	UF : 0, UT : 6,		CONFIG : 'N U T, 0, 0, 0',
	X =  493.676  mm,	Y =   -406.000  mm,	Z =   -242.674  mm,
	W =  90.000 deg,	P =   0.000 deg,	R =   90.000 deg
};
P[579]{
   GP1:
	UF : 0, UT : 6,		CONFIG : 'N U T, 0, 0, 0',
	X =  491.508  mm,	Y =   -402.493  mm,	Z =   -243.023  mm,
	W =  90.000 deg,	P =   0.000 deg,	R =   90.000 deg
};
P[580]{
   GP1:
	UF : 0, UT : 6,		CONFIG : 'N U T, 0, 0, 0',
	X =  491.035  mm,	Y =   -401.706  mm,	Z =   -243.069  mm,
	W =  90.000 deg,	P =   0.000 deg,	R =   90.000 deg
};
P[581]{
   GP1:
	UF : 0, UT : 6,		CONFIG : 'N U T, 0, 0, 0',
	X =  488.683  mm,	Y =   -397.423  mm,	Z =   -242.773  mm,
	W =  90.000 deg,	P =   0.000 deg,	R =   90.000 deg
};
P[582]{
   GP1:
	UF : 0, UT : 6,		CONFIG : 'N U T, 0, 0, 0',
	X =  487.518  mm,	Y =   -395.566  mm,	Z =   -242.999  mm,
	W =  90.000 deg,	P =   0.000 deg,	R =   90.000 deg
};
P[583]{
   GP1:
	UF : 0, UT : 6,		CONFIG : 'N U T, 0, 0, 0',
	X =  486.981  mm,	Y =   -394.534  mm,	Z =   -242.856  mm,
	W =  90.000 deg,	P =   0.000 deg,	R =   90.000 deg
};
P[584]{
   GP1:
	UF : 0, UT : 6,		CONFIG : 'N U T, 0, 0, 0',
	X =  486.353  mm,	Y =   -393.547  mm,	Z =   -242.997  mm,
	W =  90.000 deg,	P =   0.000 deg,	R =   90.000 deg
};
P[585]{
   GP1:
	UF : 0, UT : 6,		CONFIG : 'N U T, 0, 0, 0',
	X =  483.576  mm,	Y =   -388.574  mm,	Z =   -242.766  mm,
	W =  90.000 deg,	P =   0.000 deg,	R =   90.000 deg
};
P[586]{
   GP1:
	UF : 0, UT : 6,		CONFIG : 'N U T, 0, 0, 0',
	X =  482.472  mm,	Y =   -386.803  mm,	Z =   -242.966  mm,
	W =  90.000 deg,	P =   0.000 deg,	R =   90.000 deg
};
P[587]{
   GP1:
	UF : 0, UT : 6,		CONFIG : 'N U T, 0, 0, 0',
	X =  481.903  mm,	Y =   -385.635  mm,	Z =   -242.710  mm,
	W =  90.000 deg,	P =   0.000 deg,	R =   90.000 deg
};
P[588]{
   GP1:
	UF : 0, UT : 6,		CONFIG : 'N U T, 0, 0, 0',
	X =  481.173  mm,	Y =   -384.554  mm,	Z =   -242.968  mm,
	W =  90.000 deg,	P =   0.000 deg,	R =   90.000 deg
};
P[589]{
   GP1:
	UF : 0, UT : 6,		CONFIG : 'N U T, 0, 0, 0',
	X =  480.423  mm,	Y =   -383.094  mm,	Z =   -242.739  mm,
	W =  90.000 deg,	P =   0.000 deg,	R =   90.000 deg
};
P[590]{
   GP1:
	UF : 0, UT : 6,		CONFIG : 'N U T, 0, 0, 0',
	X =  479.217  mm,	Y =   -380.974  mm,	Z =   -242.697  mm,
	W =  90.000 deg,	P =   0.000 deg,	R =   90.000 deg
};
P[591]{
   GP1:
	UF : 0, UT : 6,		CONFIG : 'N U T, 0, 0, 0',
	X =  478.386  mm,	Y =   -379.549  mm,	Z =   -242.715  mm,
	W =  90.000 deg,	P =   0.000 deg,	R =   90.000 deg
};
P[592]{
   GP1:
	UF : 0, UT : 6,		CONFIG : 'N U T, 0, 0, 0',
	X =  477.243  mm,	Y =   -377.703  mm,	Z =   -242.906  mm,
	W =  90.000 deg,	P =   0.000 deg,	R =   90.000 deg
};
P[593]{
   GP1:
	UF : 0, UT : 6,		CONFIG : 'N U T, 0, 0, 0',
	X =  476.688  mm,	Y =   -376.836  mm,	Z =   -243.035  mm,
	W =  90.000 deg,	P =   0.000 deg,	R =   90.000 deg
};
P[594]{
   GP1:
	UF : 0, UT : 6,		CONFIG : 'N U T, 0, 0, 0',
	X =  475.030  mm,	Y =   -373.929  mm,	Z =   -242.986  mm,
	W =  90.000 deg,	P =   0.000 deg,	R =   90.000 deg
};
P[595]{
   GP1:
	UF : 0, UT : 6,		CONFIG : 'N U T, 0, 0, 0',
	X =  473.452  mm,	Y =   -370.951  mm,	Z =   -242.642  mm,
	W =  90.000 deg,	P =   0.000 deg,	R =   90.000 deg
};
P[596]{
   GP1:
	UF : 0, UT : 6,		CONFIG : 'N U T, 0, 0, 0',
	X =  470.449  mm,	Y =   -365.786  mm,	Z =   -242.694  mm,
	W =  90.000 deg,	P =   0.000 deg,	R =   90.000 deg
};
P[597]{
   GP1:
	UF : 0, UT : 6,		CONFIG : 'N U T, 0, 0, 0',
	X =  469.940  mm,	Y =   -364.942  mm,	Z =   -242.747  mm,
	W =  90.000 deg,	P =   0.000 deg,	R =   90.000 deg
};
P[598]{
   GP1:
	UF : 0, UT : 6,		CONFIG : 'N U T, 0, 0, 0',
	X =  469.509  mm,	Y =   -364.334  mm,	Z =   -242.939  mm,
	W =  90.000 deg,	P =   0.000 deg,	R =   90.000 deg
};
P[599]{
   GP1:
	UF : 0, UT : 6,		CONFIG : 'N U T, 0, 0, 0',
	X =  469.105  mm,	Y =   -363.483  mm,	Z =   -242.726  mm,
	W =  90.000 deg,	P =   0.000 deg,	R =   90.000 deg
};
P[600]{
   GP1:
	UF : 0, UT : 6,		CONFIG : 'N U T, 0, 0, 0',
	X =  465.819  mm,	Y =   -357.758  mm,	Z =   -242.682  mm,
	W =  90.000 deg,	P =   0.000 deg,	R =   90.000 deg
};
P[601]{
   GP1:
	UF : 0, UT : 6,		CONFIG : 'N U T, 0, 0, 0',
	X =  465.212  mm,	Y =   -356.975  mm,	Z =   -243.055  mm,
	W =  90.000 deg,	P =   0.000 deg,	R =   90.000 deg
};
P[602]{
   GP1:
	UF : 0, UT : 6,		CONFIG : 'N U T, 0, 0, 0',
	X =  464.933  mm,	Y =   -356.223  mm,	Z =   -242.679  mm,
	W =  90.000 deg,	P =   0.000 deg,	R =   90.000 deg
};
P[603]{
   GP1:
	UF : 0, UT : 6,		CONFIG : 'N U T, 0, 0, 0',
	X =  463.862  mm,	Y =   -354.544  mm,	Z =   -242.928  mm,
	W =  90.000 deg,	P =   0.000 deg,	R =   90.000 deg
};
P[604]{
   GP1:
	UF : 0, UT : 6,		CONFIG : 'N U T, 0, 0, 0',
	X =  463.227  mm,	Y =   -353.457  mm,	Z =   -242.944  mm,
	W =  90.000 deg,	P =   0.000 deg,	R =   90.000 deg
};
P[605]{
   GP1:
	UF : 0, UT : 6,		CONFIG : 'N U T, 0, 0, 0',
	X =  462.587  mm,	Y =   -352.267  mm,	Z =   -242.830  mm,
	W =  90.000 deg,	P =   0.000 deg,	R =   90.000 deg
};
P[606]{
   GP1:
	UF : 0, UT : 6,		CONFIG : 'N U T, 0, 0, 0',
	X =  461.750  mm,	Y =   -350.701  mm,	Z =   -242.669  mm,
	W =  90.000 deg,	P =   0.000 deg,	R =   90.000 deg
};
P[607]{
   GP1:
	UF : 0, UT : 6,		CONFIG : 'N U T, 0, 0, 0',
	X =  461.243  mm,	Y =   -349.841  mm,	Z =   -242.692  mm,
	W =  90.000 deg,	P =   0.000 deg,	R =   90.000 deg
};
P[608]{
   GP1:
	UF : 0, UT : 6,		CONFIG : 'N U T, 0, 0, 0',
	X =  457.667  mm,	Y =   -343.916  mm,	Z =   -243.068  mm,
	W =  90.000 deg,	P =   0.000 deg,	R =   90.000 deg
};
P[609]{
   GP1:
	UF : 0, UT : 6,		CONFIG : 'N U T, 0, 0, 0',
	X =  457.192  mm,	Y =   -342.798  mm,	Z =   -242.655  mm,
	W =  90.000 deg,	P =   0.000 deg,	R =   90.000 deg
};
P[610]{
   GP1:
	UF : 0, UT : 6,		CONFIG : 'N U T, 0, 0, 0',
	X =  456.456  mm,	Y =   -341.645  mm,	Z =   -242.825  mm,
	W =  90.000 deg,	P =   0.000 deg,	R =   90.000 deg
};
P[611]{
   GP1:
	UF : 0, UT : 6,		CONFIG : 'N U T, 0, 0, 0',
	X =  456.068  mm,	Y =   -341.111  mm,	Z =   -243.018  mm,
	W =  90.000 deg,	P =   0.000 deg,	R =   90.000 deg
};
P[612]{
   GP1:
	UF : 0, UT : 6,		CONFIG : 'N U T, 0, 0, 0',
	X =  455.729  mm,	Y =   -340.364  mm,	Z =   -242.796  mm,
	W =  90.000 deg,	P =   0.000 deg,	R =   90.000 deg
};
P[613]{
   GP1:
	UF : 0, UT : 6,		CONFIG : 'N U T, 0, 0, 0',
	X =  455.037  mm,	Y =   -339.374  mm,	Z =   -243.087  mm,
	W =  90.000 deg,	P =   0.000 deg,	R =   90.000 deg
};
P[614]{
   GP1:
	UF : 0, UT : 6,		CONFIG : 'N U T, 0, 0, 0',
	X =  454.776  mm,	Y =   -338.735  mm,	Z =   -242.825  mm,
	W =  90.000 deg,	P =   0.000 deg,	R =   90.000 deg
};
P[615]{
   GP1:
	UF : 0, UT : 6,		CONFIG : 'N U T, 0, 0, 0',
	X =  454.275  mm,	Y =   -337.758  mm,	Z =   -242.673  mm,
	W =  90.000 deg,	P =   0.000 deg,	R =   90.000 deg
};
P[616]{
   GP1:
	UF : 0, UT : 6,		CONFIG : 'N U T, 0, 0, 0',
	X =  453.418  mm,	Y =   -336.311  mm,	Z =   -242.725  mm,
	W =  90.000 deg,	P =   0.000 deg,	R =   90.000 deg
};
P[617]{
   GP1:
	UF : 0, UT : 6,		CONFIG : 'N U T, 0, 0, 0',
	X =  451.883  mm,	Y =   -333.631  mm,	Z =   -242.692  mm,
	W =  90.000 deg,	P =   0.000 deg,	R =   90.000 deg
};
P[618]{
   GP1:
	UF : 0, UT : 6,		CONFIG : 'N U T, 0, 0, 0',
	X =  450.535  mm,	Y =   -331.387  mm,	Z =   -242.820  mm,
	W =  90.000 deg,	P =   0.000 deg,	R =   90.000 deg
};
P[619]{
   GP1:
	UF : 0, UT : 6,		CONFIG : 'N U T, 0, 0, 0',
	X =  449.427  mm,	Y =   -329.483  mm,	Z =   -242.841  mm,
	W =  90.000 deg,	P =   0.000 deg,	R =   90.000 deg
};
P[620]{
   GP1:
	UF : 0, UT : 6,		CONFIG : 'N U T, 0, 0, 0',
	X =  448.882  mm,	Y =   -328.645  mm,	Z =   -242.988  mm,
	W =  90.000 deg,	P =   0.000 deg,	R =   90.000 deg
};
P[621]{
   GP1:
	UF : 0, UT : 6,		CONFIG : 'N U T, 0, 0, 0',
	X =  448.429  mm,	Y =   -327.816  mm,	Z =   -242.926  mm,
	W =  90.000 deg,	P =   0.000 deg,	R =   90.000 deg
};
P[622]{
   GP1:
	UF : 0, UT : 6,		CONFIG : 'N U T, 0, 0, 0',
	X =  447.571  mm,	Y =   -326.414  mm,	Z =   -243.046  mm,
	W =  90.000 deg,	P =   0.000 deg,	R =   90.000 deg
};
P[623]{
   GP1:
	UF : 0, UT : 6,		CONFIG : 'N U T, 0, 0, 0',
	X =  447.107  mm,	Y =   -325.501  mm,	Z =   -242.890  mm,
	W =  90.000 deg,	P =   0.000 deg,	R =   90.000 deg
};
P[624]{
   GP1:
	UF : 0, UT : 6,		CONFIG : 'N U T, 0, 0, 0',
	X =  446.125  mm,	Y =   -323.752  mm,	Z =   -242.825  mm,
	W =  90.000 deg,	P =   0.000 deg,	R =   90.000 deg
};
P[625]{
   GP1:
	UF : 0, UT : 6,		CONFIG : 'N U T, 0, 0, 0',
	X =  445.554  mm,	Y =   -322.632  mm,	Z =   -242.643  mm,
	W =  90.000 deg,	P =   0.000 deg,	R =   90.000 deg
};
P[626]{
   GP1:
	UF : 0, UT : 6,		CONFIG : 'N U T, 0, 0, 0',
	X =  445.043  mm,	Y =   -322.036  mm,	Z =   -243.046  mm,
	W =  90.000 deg,	P =   0.000 deg,	R =   90.000 deg
};
P[627]{
   GP1:
	UF : 0, UT : 6,		CONFIG : 'N U T, 0, 0, 0',
	X =  444.429  mm,	Y =   -320.723  mm,	Z =   -242.695  mm,
	W =  90.000 deg,	P =   0.000 deg,	R =   90.000 deg
};
P[628]{
   GP1:
	UF : 0, UT : 6,		CONFIG : 'N U T, 0, 0, 0',
	X =  443.256  mm,	Y =   -318.924  mm,	Z =   -243.022  mm,
	W =  90.000 deg,	P =   0.000 deg,	R =   90.000 deg
};
P[629]{
   GP1:
	UF : 0, UT : 6,		CONFIG : 'N U T, 0, 0, 0',
	X =  442.402  mm,	Y =   -317.399  mm,	Z =   -242.957  mm,
	W =  90.000 deg,	P =   0.000 deg,	R =   90.000 deg
};
P[630]{
   GP1:
	UF : 0, UT : 6,		CONFIG : 'N U T, 0, 0, 0',
	X =  441.806  mm,	Y =   -316.199  mm,	Z =   -242.722  mm,
	W =  90.000 deg,	P =   0.000 deg,	R =   90.000 deg
};
P[631]{
   GP1:
	UF : 0, UT : 6,		CONFIG : 'N U T, 0, 0, 0',
	X =  440.252  mm,	Y =   -313.727  mm,	Z =   -243.029  mm,
	W =  90.000 deg,	P =   0.000 deg,	R =   90.000 deg
};
P[632]{
   GP1:
	UF : 0, UT : 6,		CONFIG : 'N U T, 0, 0, 0',
	X =  439.890  mm,	Y =   -312.921  mm,	Z =   -242.779  mm,
	W =  90.000 deg,	P =   0.000 deg,	R =   90.000 deg
};
P[633]{
   GP1:
	UF : 0, UT : 6,		CONFIG : 'N U T, 0, 0, 0',
	X =  437.698  mm,	Y =   -309.288  mm,	Z =   -243.010  mm,
	W =  90.000 deg,	P =   0.000 deg,	R =   90.000 deg
};
P[634]{
   GP1:
	UF : 0, UT : 6,		CONFIG : 'N U T, 0, 0, 0',
	X =  436.916  mm,	Y =   -307.753  mm,	Z =   -242.754  mm,
	W =  90.000 deg,	P =   0.000 deg,	R =   90.000 deg
};
P[635]{
   GP1:
	UF : 0, UT : 6,		CONFIG : 'N U T, 0, 0, 0',
	X =  436.415  mm,	Y =   -306.911  mm,	Z =   -242.791  mm,
	W =  90.000 deg,	P =   0.000 deg,	R =   90.000 deg
};
P[636]{
   GP1:
	UF : 0, UT : 6,		CONFIG : 'N U T, 0, 0, 0',
	X =  434.702  mm,	Y =   -303.882  mm,	Z =   -242.703  mm,
	W =  90.000 deg,	P =   0.000 deg,	R =   90.000 deg
};
P[637]{
   GP1:
	UF : 0, UT : 6,		CONFIG : 'N U T, 0, 0, 0',
	X =  433.644  mm,	Y =   -302.168  mm,	Z =   -242.871  mm,
	W =  90.000 deg,	P =   0.000 deg,	R =   90.000 deg
};
P[638]{
   GP1:
	UF : 0, UT : 6,		CONFIG : 'N U T, 0, 0, 0',
	X =  432.712  mm,	Y =   -300.683  mm,	Z =   -243.050  mm,
	W =  90.000 deg,	P =   0.000 deg,	R =   90.000 deg
};
P[639]{
   GP1:
	UF : 0, UT : 6,		CONFIG : 'N U T, 0, 0, 0',
	X =  432.248  mm,	Y =   -299.846  mm,	Z =   -243.004  mm,
	W =  90.000 deg,	P =   0.000 deg,	R =   90.000 deg
};
P[640]{
   GP1:
	UF : 0, UT : 6,		CONFIG : 'N U T, 0, 0, 0',
	X =  431.048  mm,	Y =   -297.523  mm,	Z =   -242.659  mm,
	W =  90.000 deg,	P =   0.000 deg,	R =   90.000 deg
};
P[641]{
   GP1:
	UF : 0, UT : 6,		CONFIG : 'N U T, 0, 0, 0',
	X =  430.193  mm,	Y =   -296.056  mm,	Z =   -242.681  mm,
	W =  90.000 deg,	P =   0.000 deg,	R =   90.000 deg
};
P[642]{
   GP1:
	UF : 0, UT : 6,		CONFIG : 'N U T, 0, 0, 0',
	X =  429.186  mm,	Y =   -294.339  mm,	Z =   -242.719  mm,
	W =  90.000 deg,	P =   0.000 deg,	R =   90.000 deg
};
P[643]{
   GP1:
	UF : 0, UT : 6,		CONFIG : 'N U T, 0, 0, 0',
	X =  428.670  mm,	Y =   -293.571  mm,	Z =   -242.895  mm,
	W =  90.000 deg,	P =   0.000 deg,	R =   90.000 deg
};
P[644]{
   GP1:
	UF : 0, UT : 6,		CONFIG : 'N U T, 0, 0, 0',
	X =  427.766  mm,	Y =   -291.900  mm,	Z =   -242.749  mm,
	W =  90.000 deg,	P =   0.000 deg,	R =   90.000 deg
};
P[645]{
   GP1:
	UF : 0, UT : 6,		CONFIG : 'N U T, 0, 0, 0',
	X =  427.262  mm,	Y =   -291.213  mm,	Z =   -243.007  mm,
	W =  90.000 deg,	P =   0.000 deg,	R =   90.000 deg
};
P[646]{
   GP1:
	UF : 0, UT : 6,		CONFIG : 'N U T, 0, 0, 0',
	X =  425.850  mm,	Y =   -288.767  mm,	Z =   -243.006  mm,
	W =  90.000 deg,	P =   0.000 deg,	R =   90.000 deg
};
P[647]{
   GP1:
	UF : 0, UT : 6,		CONFIG : 'N U T, 0, 0, 0',
	X =  424.872  mm,	Y =   -286.842  mm,	Z =   -242.684  mm,
	W =  90.000 deg,	P =   0.000 deg,	R =   90.000 deg
};
P[648]{
   GP1:
	UF : 0, UT : 6,		CONFIG : 'N U T, 0, 0, 0',
	X =  424.478  mm,	Y =   -286.472  mm,	Z =   -243.120  mm,
	W =  90.000 deg,	P =   0.000 deg,	R =   90.000 deg
};
P[649]{
   GP1:
	UF : 0, UT : 6,		CONFIG : 'N U T, 0, 0, 0',
	X =  424.033  mm,	Y =   -285.395  mm,	Z =   -242.689  mm,
	W =  90.000 deg,	P =   0.000 deg,	R =   90.000 deg
};
P[650]{
   GP1:
	UF : 0, UT : 6,		CONFIG : 'N U T, 0, 0, 0',
	X =  423.488  mm,	Y =   -284.533  mm,	Z =   -242.808  mm,
	W =  90.000 deg,	P =   0.000 deg,	R =   90.000 deg
};
P[651]{
   GP1:
	UF : 0, UT : 6,		CONFIG : 'N U T, 0, 0, 0',
	X =  422.717  mm,	Y =   -283.361  mm,	Z =   -243.036  mm,
	W =  90.000 deg,	P =   0.000 deg,	R =   90.000 deg
};
P[652]{
   GP1:
	UF : 0, UT : 6,		CONFIG : 'N U T, 0, 0, 0',
	X =  420.867  mm,	Y =   -280.066  mm,	Z =   -242.906  mm,
	W =  90.000 deg,	P =   0.000 deg,	R =   90.000 deg
};
P[653]{
   GP1:
	UF : 0, UT : 6,		CONFIG : 'N U T, 0, 0, 0',
	X =  420.362  mm,	Y =   -279.074  mm,	Z =   -242.741  mm,
	W =  90.000 deg,	P =   0.000 deg,	R =   90.000 deg
};
P[654]{
   GP1:
	UF : 0, UT : 6,		CONFIG : 'N U T, 0, 0, 0',
	X =  419.112  mm,	Y =   -276.985  mm,	Z =   -242.851  mm,
	W =  90.000 deg,	P =   0.000 deg,	R =   90.000 deg
};
P[655]{
   GP1:
	UF : 0, UT : 6,		CONFIG : 'N U T, 0, 0, 0',
	X =  416.395  mm,	Y =   -272.218  mm,	Z =   -242.762  mm,
	W =  90.000 deg,	P =   0.000 deg,	R =   90.000 deg
};
P[656]{
   GP1:
	UF : 0, UT : 6,		CONFIG : 'N U T, 0, 0, 0',
	X =  415.347  mm,	Y =   -270.532  mm,	Z =   -242.946  mm,
	W =  90.000 deg,	P =   0.000 deg,	R =   90.000 deg
};
P[657]{
   GP1:
	UF : 0, UT : 6,		CONFIG : 'N U T, 0, 0, 0',
	X =  414.972  mm,	Y =   -269.687  mm,	Z =   -242.669  mm,
	W =  90.000 deg,	P =   0.000 deg,	R =   90.000 deg
};
P[658]{
   GP1:
	UF : 0, UT : 6,		CONFIG : 'N U T, 0, 0, 0',
	X =  412.304  mm,	Y =   -265.079  mm,	Z =   -242.689  mm,
	W =  90.000 deg,	P =   0.000 deg,	R =   90.000 deg
};
P[659]{
   GP1:
	UF : 0, UT : 6,		CONFIG : 'N U T, 0, 0, 0',
	X =  409.893  mm,	Y =   -261.017  mm,	Z =   -242.849  mm,
	W =  90.000 deg,	P =   0.000 deg,	R =   90.000 deg
};
P[660]{
   GP1:
	UF : 0, UT : 6,		CONFIG : 'N U T, 0, 0, 0',
	X =  408.519  mm,	Y =   -258.620  mm,	Z =   -242.823  mm,
	W =  90.000 deg,	P =   0.000 deg,	R =   90.000 deg
};
P[661]{
   GP1:
	UF : 0, UT : 6,		CONFIG : 'N U T, 0, 0, 0',
	X =  407.948  mm,	Y =   -257.573  mm,	Z =   -242.742  mm,
	W =  90.000 deg,	P =   0.000 deg,	R =   90.000 deg
};
P[662]{
   GP1:
	UF : 0, UT : 6,		CONFIG : 'N U T, 0, 0, 0',
	X =  406.916  mm,	Y =   -255.724  mm,	Z =   -242.656  mm,
	W =  90.000 deg,	P =   0.000 deg,	R =   90.000 deg
};
P[663]{
   GP1:
	UF : 0, UT : 6,		CONFIG : 'N U T, 0, 0, 0',
	X =  406.248  mm,	Y =   -254.717  mm,	Z =   -242.866  mm,
	W =  90.000 deg,	P =   0.000 deg,	R =   90.000 deg
};
P[664]{
   GP1:
	UF : 0, UT : 6,		CONFIG : 'N U T, 0, 0, 0',
	X =  405.826  mm,	Y =   -254.148  mm,	Z =   -243.094  mm,
	W =  90.000 deg,	P =   0.000 deg,	R =   90.000 deg
};
P[665]{
   GP1:
	UF : 0, UT : 6,		CONFIG : 'N U T, 0, 0, 0',
	X =  405.359  mm,	Y =   -253.014  mm,	Z =   -242.636  mm,
	W =  90.000 deg,	P =   0.000 deg,	R =   90.000 deg
};
P[666]{
   GP1:
	UF : 0, UT : 6,		CONFIG : 'N U T, 0, 0, 0',
	X =  404.831  mm,	Y =   -252.283  mm,	Z =   -242.895  mm,
	W =  90.000 deg,	P =   0.000 deg,	R =   90.000 deg
};
P[667]{
   GP1:
	UF : 0, UT : 6,		CONFIG : 'N U T, 0, 0, 0',
	X =  404.404  mm,	Y =   -251.542  mm,	Z =   -242.890  mm,
	W =  90.000 deg,	P =   0.000 deg,	R =   90.000 deg
};
P[668]{
   GP1:
	UF : 0, UT : 6,		CONFIG : 'N U T, 0, 0, 0',
	X =  404.048  mm,	Y =   -250.852  mm,	Z =   -242.788  mm,
	W =  90.000 deg,	P =   0.000 deg,	R =   90.000 deg
};
P[669]{
   GP1:
	UF : 0, UT : 6,		CONFIG : 'N U T, 0, 0, 0',
	X =  403.086  mm,	Y =   -249.200  mm,	Z =   -242.808  mm,
	W =  90.000 deg,	P =   0.000 deg,	R =   90.000 deg
};
P[670]{
   GP1:
	UF : 0, UT : 6,		CONFIG : 'N U T, 0, 0, 0',
	X =  402.241  mm,	Y =   -247.854  mm,	Z =   -242.974  mm,
	W =  90.000 deg,	P =   0.000 deg,	R =   90.000 deg
};
P[671]{
   GP1:
	UF : 0, UT : 6,		CONFIG : 'N U T, 0, 0, 0',
	X =  401.722  mm,	Y =   -246.786  mm,	Z =   -242.735  mm,
	W =  90.000 deg,	P =   0.000 deg,	R =   90.000 deg
};
P[672]{
   GP1:
	UF : 0, UT : 6,		CONFIG : 'N U T, 0, 0, 0',
	X =  400.136  mm,	Y =   -244.140  mm,	Z =   -242.874  mm,
	W =  90.000 deg,	P =   0.000 deg,	R =   90.000 deg
};
P[673]{
   GP1:
	UF : 0, UT : 6,		CONFIG : 'N U T, 0, 0, 0',
	X =  399.693  mm,	Y =   -243.411  mm,	Z =   -242.932  mm,
	W =  90.000 deg,	P =   0.000 deg,	R =   90.000 deg
};
P[674]{
   GP1:
	UF : 0, UT : 6,		CONFIG : 'N U T, 0, 0, 0',
	X =  399.160  mm,	Y =   -242.303  mm,	Z =   -242.673  mm,
	W =  90.000 deg,	P =   0.000 deg,	R =   90.000 deg
};
P[675]{
   GP1:
	UF : 0, UT : 6,		CONFIG : 'N U T, 0, 0, 0',
	X =  398.016  mm,	Y =   -240.433  mm,	Z =   -242.828  mm,
	W =  90.000 deg,	P =   0.000 deg,	R =   90.000 deg
};
P[676]{
   GP1:
	UF : 0, UT : 6,		CONFIG : 'N U T, 0, 0, 0',
	X =  396.958  mm,	Y =   -238.670  mm,	Z =   -242.926  mm,
	W =  90.000 deg,	P =   0.000 deg,	R =   90.000 deg
};
P[677]{
   GP1:
	UF : 0, UT : 6,		CONFIG : 'N U T, 0, 0, 0',
	X =  396.580  mm,	Y =   -237.820  mm,	Z =   -242.651  mm,
	W =  90.000 deg,	P =   0.000 deg,	R =   90.000 deg
};
P[678]{
   GP1:
	UF : 0, UT : 6,		CONFIG : 'N U T, 0, 0, 0',
	X =  395.962  mm,	Y =   -236.968  mm,	Z =   -242.958  mm,
	W =  90.000 deg,	P =   0.000 deg,	R =   90.000 deg
};
P[679]{
   GP1:
	UF : 0, UT : 6,		CONFIG : 'N U T, 0, 0, 0',
	X =  393.838  mm,	Y =   -233.256  mm,	Z =   -242.912  mm,
	W =  90.000 deg,	P =   0.000 deg,	R =   90.000 deg
};
P[680]{
   GP1:
	UF : 0, UT : 6,		CONFIG : 'N U T, 0, 0, 0',
	X =  393.402  mm,	Y =   -232.479  mm,	Z =   -242.879  mm,
	W =  90.000 deg,	P =   0.000 deg,	R =   90.000 deg
};
P[681]{
   GP1:
	UF : 0, UT : 6,		CONFIG : 'N U T, 0, 0, 0',
	X =  392.843  mm,	Y =   -231.497  mm,	Z =   -242.860  mm,
	W =  90.000 deg,	P =   0.000 deg,	R =   90.000 deg
};
P[682]{
   GP1:
	UF : 0, UT : 6,		CONFIG : 'N U T, 0, 0, 0',
	X =  392.529  mm,	Y =   -230.816  mm,	Z =   -242.669  mm,
	W =  90.000 deg,	P =   0.000 deg,	R =   90.000 deg
};
P[683]{
   GP1:
	UF : 0, UT : 6,		CONFIG : 'N U T, 0, 0, 0',
	X =  391.298  mm,	Y =   -228.806  mm,	Z =   -242.841  mm,
	W =  90.000 deg,	P =   0.000 deg,	R =   90.000 deg
};
P[684]{
   GP1:
	UF : 0, UT : 6,		CONFIG : 'N U T, 0, 0, 0',
	X =  390.549  mm,	Y =   -227.710  mm,	Z =   -243.121  mm,
	W =  90.000 deg,	P =   0.000 deg,	R =   90.000 deg
};
P[685]{
   GP1:
	UF : 0, UT : 6,		CONFIG : 'N U T, 0, 0, 0',
	X =  389.062  mm,	Y =   -224.820  mm,	Z =   -242.680  mm,
	W =  90.000 deg,	P =   0.000 deg,	R =   90.000 deg
};
P[686]{
   GP1:
	UF : 0, UT : 6,		CONFIG : 'N U T, 0, 0, 0',
	X =  388.423  mm,	Y =   -223.763  mm,	Z =   -242.749  mm,
	W =  90.000 deg,	P =   0.000 deg,	R =   90.000 deg
};
P[687]{
   GP1:
	UF : 0, UT : 6,		CONFIG : 'N U T, 0, 0, 0',
	X =  387.709  mm,	Y =   -222.537  mm,	Z =   -242.765  mm,
	W =  90.000 deg,	P =   0.000 deg,	R =   90.000 deg
};
P[688]{
   GP1:
	UF : 0, UT : 6,		CONFIG : 'N U T, 0, 0, 0',
	X =  386.978  mm,	Y =   -221.353  mm,	Z =   -242.880  mm,
	W =  90.000 deg,	P =   0.000 deg,	R =   90.000 deg
};
P[689]{
   GP1:
	UF : 0, UT : 6,		CONFIG : 'N U T, 0, 0, 0',
	X =  386.062  mm,	Y =   -219.686  mm,	Z =   -242.765  mm,
	W =  90.000 deg,	P =   0.000 deg,	R =   90.000 deg
};
P[690]{
   GP1:
	UF : 0, UT : 6,		CONFIG : 'N U T, 0, 0, 0',
	X =  384.657  mm,	Y =   -217.491  mm,	Z =   -243.101  mm,
	W =  90.000 deg,	P =   0.000 deg,	R =   90.000 deg
};
P[691]{
   GP1:
	UF : 0, UT : 6,		CONFIG : 'N U T, 0, 0, 0',
	X =  384.296  mm,	Y =   -216.555  mm,	Z =   -242.666  mm,
	W =  90.000 deg,	P =   0.000 deg,	R =   90.000 deg
};
P[692]{
   GP1:
	UF : 0, UT : 6,		CONFIG : 'N U T, 0, 0, 0',
	X =  383.451  mm,	Y =   -215.130  mm,	Z =   -242.720  mm,
	W =  90.000 deg,	P =   0.000 deg,	R =   90.000 deg
};
P[693]{
   GP1:
	UF : 0, UT : 6,		CONFIG : 'N U T, 0, 0, 0',
	X =  383.107  mm,	Y =   -214.511  mm,	Z =   -242.687  mm,
	W =  90.000 deg,	P =   0.000 deg,	R =   90.000 deg
};
P[694]{
   GP1:
	UF : 0, UT : 6,		CONFIG : 'N U T, 0, 0, 0',
	X =  382.431  mm,	Y =   -213.381  mm,	Z =   -242.743  mm,
	W =  90.000 deg,	P =   0.000 deg,	R =   90.000 deg
};
P[695]{
   GP1:
	UF : 0, UT : 6,		CONFIG : 'N U T, 0, 0, 0',
	X =  381.118  mm,	Y =   -211.223  mm,	Z =   -242.906  mm,
	W =  90.000 deg,	P =   0.000 deg,	R =   90.000 deg
};
P[696]{
   GP1:
	UF : 0, UT : 6,		CONFIG : 'N U T, 0, 0, 0',
	X =  380.507  mm,	Y =   -210.010  mm,	Z =   -242.688  mm,
	W =  90.000 deg,	P =   0.000 deg,	R =   90.000 deg
};
P[697]{
   GP1:
	UF : 0, UT : 6,		CONFIG : 'N U T, 0, 0, 0',
	X =  379.547  mm,	Y =   -208.506  mm,	Z =   -242.911  mm,
	W =  90.000 deg,	P =   0.000 deg,	R =   90.000 deg
};
P[698]{
   GP1:
	UF : 0, UT : 6,		CONFIG : 'N U T, 0, 0, 0',
	X =  379.110  mm,	Y =   -207.893  mm,	Z =   -243.113  mm,
	W =  90.000 deg,	P =   0.000 deg,	R =   90.000 deg
};
P[699]{
   GP1:
	UF : 0, UT : 6,		CONFIG : 'N U T, 0, 0, 0',
	X =  378.865  mm,	Y =   -207.199  mm,	Z =   -242.735  mm,
	W =  90.000 deg,	P =   0.000 deg,	R =   90.000 deg
};
P[700]{
   GP1:
	UF : 0, UT : 6,		CONFIG : 'N U T, 0, 0, 0',
	X =  378.410  mm,	Y =   -206.373  mm,	Z =   -242.681  mm,
	W =  90.000 deg,	P =   0.000 deg,	R =   90.000 deg
};
P[701]{
   GP1:
	UF : 0, UT : 6,		CONFIG : 'N U T, 0, 0, 0',
	X =  377.950  mm,	Y =   -205.566  mm,	Z =   -242.669  mm,
	W =  90.000 deg,	P =   0.000 deg,	R =   90.000 deg
};
P[702]{
   GP1:
	UF : 0, UT : 6,		CONFIG : 'N U T, 0, 0, 0',
	X =  377.118  mm,	Y =   -204.305  mm,	Z =   -242.919  mm,
	W =  90.000 deg,	P =   0.000 deg,	R =   90.000 deg
};
P[703]{
   GP1:
	UF : 0, UT : 6,		CONFIG : 'N U T, 0, 0, 0',
	X =  376.300  mm,	Y =   -202.770  mm,	Z =   -242.755  mm,
	W =  90.000 deg,	P =   0.000 deg,	R =   90.000 deg
};
P[704]{
   GP1:
	UF : 0, UT : 6,		CONFIG : 'N U T, 0, 0, 0',
	X =  375.677  mm,	Y =   -201.626  mm,	Z =   -242.661  mm,
	W =  90.000 deg,	P =   0.000 deg,	R =   90.000 deg
};
P[705]{
   GP1:
	UF : 0, UT : 6,		CONFIG : 'N U T, 0, 0, 0',
	X =  374.613  mm,	Y =   -199.790  mm,	Z =   -242.674  mm,
	W =  90.000 deg,	P =   0.000 deg,	R =   90.000 deg
};
P[706]{
   GP1:
	UF : 0, UT : 6,		CONFIG : 'N U T, 0, 0, 0',
	X =  373.340  mm,	Y =   -197.859  mm,	Z =   -243.057  mm,
	W =  90.000 deg,	P =   0.000 deg,	R =   90.000 deg
};
P[707]{
   GP1:
	UF : 0, UT : 6,		CONFIG : 'N U T, 0, 0, 0',
	X =  372.811  mm,	Y =   -196.679  mm,	Z =   -242.688  mm,
	W =  90.000 deg,	P =   0.000 deg,	R =   90.000 deg
};
P[708]{
   GP1:
	UF : 0, UT : 6,		CONFIG : 'N U T, 0, 0, 0',
	X =  371.605  mm,	Y =   -194.658  mm,	Z =   -242.780  mm,
	W =  90.000 deg,	P =   0.000 deg,	R =   90.000 deg
};
P[709]{
   GP1:
	UF : 0, UT : 6,		CONFIG : 'N U T, 0, 0, 0',
	X =  371.081  mm,	Y =   -193.975  mm,	Z =   -243.096  mm,
	W =  90.000 deg,	P =   0.000 deg,	R =   90.000 deg
};
P[710]{
   GP1:
	UF : 0, UT : 6,		CONFIG : 'N U T, 0, 0, 0',
	X =  370.429  mm,	Y =   -192.649  mm,	Z =   -242.822  mm,
	W =  90.000 deg,	P =   0.000 deg,	R =   90.000 deg
};
P[711]{
   GP1:
	UF : 0, UT : 6,		CONFIG : 'N U T, 0, 0, 0',
	X =  369.848  mm,	Y =   -191.853  mm,	Z =   -243.114  mm,
	W =  90.000 deg,	P =   0.000 deg,	R =   90.000 deg
};
P[712]{
   GP1:
	UF : 0, UT : 6,		CONFIG : 'N U T, 0, 0, 0',
	X =  368.333  mm,	Y =   -188.909  mm,	Z =   -242.668  mm,
	W =  90.000 deg,	P =   0.000 deg,	R =   90.000 deg
};
P[713]{
   GP1:
	UF : 0, UT : 6,		CONFIG : 'N U T, 0, 0, 0',
	X =  366.824  mm,	Y =   -186.415  mm,	Z =   -242.834  mm,
	W =  90.000 deg,	P =   0.000 deg,	R =   90.000 deg
};
P[714]{
   GP1:
	UF : 0, UT : 6,		CONFIG : 'N U T, 0, 0, 0',
	X =  364.611  mm,	Y =   -182.483  mm,	Z =   -242.697  mm,
	W =  90.000 deg,	P =   0.000 deg,	R =   90.000 deg
};
P[715]{
   GP1:
	UF : 0, UT : 6,		CONFIG : 'N U T, 0, 0, 0',
	X =  363.673  mm,	Y =   -180.920  mm,	Z =   -242.781  mm,
	W =  90.000 deg,	P =   0.000 deg,	R =   90.000 deg
};
P[716]{
   GP1:
	UF : 0, UT : 6,		CONFIG : 'N U T, 0, 0, 0',
	X =  362.755  mm,	Y =   -179.328  mm,	Z =   -242.778  mm,
	W =  90.000 deg,	P =   0.000 deg,	R =   90.000 deg
};
P[717]{
   GP1:
	UF : 0, UT : 6,		CONFIG : 'N U T, 0, 0, 0',
	X =  361.711  mm,	Y =   -177.460  mm,	Z =   -242.694  mm,
	W =  90.000 deg,	P =   0.000 deg,	R =   90.000 deg
};
P[718]{
   GP1:
	UF : 0, UT : 6,		CONFIG : 'N U T, 0, 0, 0',
	X =  360.906  mm,	Y =   -176.081  mm,	Z =   -242.714  mm,
	W =  90.000 deg,	P =   0.000 deg,	R =   90.000 deg
};
P[719]{
   GP1:
	UF : 0, UT : 6,		CONFIG : 'N U T, 0, 0, 0',
	X =  359.562  mm,	Y =   -173.838  mm,	Z =   -242.833  mm,
	W =  90.000 deg,	P =   0.000 deg,	R =   90.000 deg
};
P[720]{
   GP1:
	UF : 0, UT : 6,		CONFIG : 'N U T, 0, 0, 0',
	X =  358.611  mm,	Y =   -172.124  mm,	Z =   -242.740  mm,
	W =  90.000 deg,	P =   0.000 deg,	R =   90.000 deg
};
P[721]{
   GP1:
	UF : 0, UT : 6,		CONFIG : 'N U T, 0, 0, 0',
	X =  357.614  mm,	Y =   -170.364  mm,	Z =   -242.694  mm,
	W =  90.000 deg,	P =   0.000 deg,	R =   90.000 deg
};
P[722]{
   GP1:
	UF : 0, UT : 6,		CONFIG : 'N U T, 0, 0, 0',
	X =  356.802  mm,	Y =   -168.935  mm,	Z =   -242.661  mm,
	W =  90.000 deg,	P =   0.000 deg,	R =   90.000 deg
};
P[723]{
   GP1:
	UF : 0, UT : 6,		CONFIG : 'N U T, 0, 0, 0',
	X =  355.568  mm,	Y =   -166.877  mm,	Z =   -242.773  mm,
	W =  90.000 deg,	P =   0.000 deg,	R =   90.000 deg
};
P[724]{
   GP1:
	UF : 0, UT : 6,		CONFIG : 'N U T, 0, 0, 0',
	X =  355.009  mm,	Y =   -165.920  mm,	Z =   -242.789  mm,
	W =  90.000 deg,	P =   0.000 deg,	R =   90.000 deg
};
P[725]{
   GP1:
	UF : 0, UT : 6,		CONFIG : 'N U T, 0, 0, 0',
	X =  354.326  mm,	Y =   -164.949  mm,	Z =   -243.087  mm,
	W =  90.000 deg,	P =   0.000 deg,	R =   90.000 deg
};
P[726]{
   GP1:
	UF : 0, UT : 6,		CONFIG : 'N U T, 0, 0, 0',
	X =  351.756  mm,	Y =   -160.324  mm,	Z =   -242.842  mm,
	W =  90.000 deg,	P =   0.000 deg,	R =   90.000 deg
};
P[727]{
   GP1:
	UF : 0, UT : 6,		CONFIG : 'N U T, 0, 0, 0',
	X =  351.206  mm,	Y =   -159.373  mm,	Z =   -242.845  mm,
	W =  90.000 deg,	P =   0.000 deg,	R =   90.000 deg
};
P[728]{
   GP1:
	UF : 0, UT : 6,		CONFIG : 'N U T, 0, 0, 0',
	X =  350.306  mm,	Y =   -157.726  mm,	Z =   -242.721  mm,
	W =  90.000 deg,	P =   0.000 deg,	R =   90.000 deg
};
P[729]{
   GP1:
	UF : 0, UT : 6,		CONFIG : 'N U T, 0, 0, 0',
	X =  349.094  mm,	Y =   -155.861  mm,	Z =   -243.047  mm,
	W =  90.000 deg,	P =   0.000 deg,	R =   90.000 deg
};
P[730]{
   GP1:
	UF : 0, UT : 6,		CONFIG : 'N U T, 0, 0, 0',
	X =  347.675  mm,	Y =   -153.166  mm,	Z =   -242.716  mm,
	W =  90.000 deg,	P =   0.000 deg,	R =   90.000 deg
};
P[731]{
   GP1:
	UF : 0, UT : 6,		CONFIG : 'N U T, 0, 0, 0',
	X =  347.111  mm,	Y =   -152.157  mm,	Z =   -242.669  mm,
	W =  90.000 deg,	P =   0.000 deg,	R =   90.000 deg
};
P[732]{
   GP1:
	UF : 0, UT : 6,		CONFIG : 'N U T, 0, 0, 0',
	X =  346.783  mm,	Y =   -151.677  mm,	Z =   -242.793  mm,
	W =  90.000 deg,	P =   0.000 deg,	R =   90.000 deg
};
P[733]{
   GP1:
	UF : 0, UT : 6,		CONFIG : 'N U T, 0, 0, 0',
	X =  344.235  mm,	Y =   -147.313  mm,	Z =   -242.863  mm,
	W =  90.000 deg,	P =   0.000 deg,	R =   90.000 deg
};
P[734]{
   GP1:
	UF : 0, UT : 6,		CONFIG : 'N U T, 0, 0, 0',
	X =  343.543  mm,	Y =   -146.004  mm,	Z =   -242.707  mm,
	W =  90.000 deg,	P =   0.000 deg,	R =   90.000 deg
};
P[735]{
   GP1:
	UF : 0, UT : 6,		CONFIG : 'N U T, 0, 0, 0',
	X =  342.929  mm,	Y =   -144.968  mm,	Z =   -242.744  mm,
	W =  90.000 deg,	P =   0.000 deg,	R =   90.000 deg
};
P[736]{
   GP1:
	UF : 0, UT : 6,		CONFIG : 'N U T, 0, 0, 0',
	X =  342.270  mm,	Y =   -144.073  mm,	Z =   -242.928  mm,
	W =  90.000 deg,	P =   0.000 deg,	R =   90.000 deg
};
P[737]{
   GP1:
	UF : 0, UT : 6,		CONFIG : 'N U T, 0, 0, 0',
	X =  340.476  mm,	Y =   -141.770  mm,	Z =   -242.882  mm,
	W =  90.000 deg,	P =   0.000 deg,	R =   90.000 deg
};
P[738]{
   GP1:
	UF : 0, UT : 6,		CONFIG : 'N U T, 0, 0, 0',
	X =  340.043  mm,	Y =   -141.280  mm,	Z =   -242.701  mm,
	W =  90.000 deg,	P =   0.000 deg,	R =   90.000 deg
};
P[739]{
   GP1:
	UF : 0, UT : 6,		CONFIG : 'N U T, 0, 0, 0',
	X =  338.981  mm,	Y =   -140.584  mm,	Z =   -243.096  mm,
	W =  90.000 deg,	P =   0.000 deg,	R =   90.000 deg
};
P[740]{
   GP1:
	UF : 0, UT : 6,		CONFIG : 'N U T, 0, 0, 0',
	X =  338.212  mm,	Y =   -139.866  mm,	Z =   -242.756  mm,
	W =  90.000 deg,	P =   0.000 deg,	R =   90.000 deg
};
P[741]{
   GP1:
	UF : 0, UT : 6,		CONFIG : 'N U T, 0, 0, 0',
	X =  336.057  mm,	Y =   -138.822  mm,	Z =   -242.877  mm,
	W =  90.000 deg,	P =   0.000 deg,	R =   90.000 deg
};
P[742]{
   GP1:
	UF : 0, UT : 6,		CONFIG : 'N U T, 0, 0, 0',
	X =  334.942  mm,	Y =   -138.549  mm,	Z =   -242.970  mm,
	W =  90.000 deg,	P =   0.000 deg,	R =   90.000 deg
};
P[743]{
   GP1:
	UF : 0, UT : 6,		CONFIG : 'N U T, 0, 0, 0',
	X =  333.776  mm,	Y =   -138.079  mm,	Z =   -242.656  mm,
	W =  90.000 deg,	P =   0.000 deg,	R =   90.000 deg
};
P[744]{
   GP1:
	UF : 0, UT : 6,		CONFIG : 'N U T, 0, 0, 0',
	X =  332.452  mm,	Y =   -137.945  mm,	Z =   -242.644  mm,
	W =  90.000 deg,	P =   0.000 deg,	R =   90.000 deg
};
P[745]{
   GP1:
	UF : 0, UT : 6,		CONFIG : 'N U T, 0, 0, 0',
	X =  330.010  mm,	Y =   -138.093  mm,	Z =   -242.840  mm,
	W =  90.000 deg,	P =   0.000 deg,	R =   90.000 deg
};
P[746]{
   GP1:
	UF : 0, UT : 6,		CONFIG : 'N U T, 0, 0, 0',
	X =  329.383  mm,	Y =   -138.234  mm,	Z =   -242.869  mm,
	W =  90.000 deg,	P =   0.000 deg,	R =   90.000 deg
};
P[747]{
   GP1:
	UF : 0, UT : 6,		CONFIG : 'N U T, 0, 0, 0',
	X =  328.708  mm,	Y =   -138.405  mm,	Z =   -242.947  mm,
	W =  90.000 deg,	P =   0.000 deg,	R =   90.000 deg
};
P[748]{
   GP1:
	UF : 0, UT : 6,		CONFIG : 'N U T, 0, 0, 0',
	X =  327.477  mm,	Y =   -138.612  mm,	Z =   -242.680  mm,
	W =  90.000 deg,	P =   0.000 deg,	R =   90.000 deg
};
P[749]{
   GP1:
	UF : 0, UT : 6,		CONFIG : 'N U T, 0, 0, 0',
	X =  326.448  mm,	Y =   -139.148  mm,	Z =   -242.924  mm,
	W =  90.000 deg,	P =   0.000 deg,	R =   90.000 deg
};
P[750]{
   GP1:
	UF : 0, UT : 6,		CONFIG : 'N U T, 0, 0, 0',
	X =  323.845  mm,	Y =   -140.474  mm,	Z =   -242.970  mm,
	W =  90.000 deg,	P =   0.000 deg,	R =   90.000 deg
};
P[751]{
   GP1:
	UF : 0, UT : 6,		CONFIG : 'N U T, 0, 0, 0',
	X =  322.599  mm,	Y =   -141.095  mm,	Z =   -242.733  mm,
	W =  90.000 deg,	P =   0.000 deg,	R =   90.000 deg
};
P[752]{
   GP1:
	UF : 0, UT : 6,		CONFIG : 'N U T, 0, 0, 0',
	X =  321.928  mm,	Y =   -141.560  mm,	Z =   -242.920  mm,
	W =  90.000 deg,	P =   0.000 deg,	R =   90.000 deg
};
P[753]{
   GP1:
	UF : 0, UT : 6,		CONFIG : 'N U T, 0, 0, 0',
	X =  320.900  mm,	Y =   -142.105  mm,	Z =   -242.802  mm,
	W =  90.000 deg,	P =   0.000 deg,	R =   90.000 deg
};
P[754]{
   GP1:
	UF : 0, UT : 6,		CONFIG : 'N U T, 0, 0, 0',
	X =  318.687  mm,	Y =   -143.403  mm,	Z =   -242.851  mm,
	W =  90.000 deg,	P =   0.000 deg,	R =   90.000 deg
};
P[755]{
   GP1:
	UF : 0, UT : 6,		CONFIG : 'N U T, 0, 0, 0',
	X =  317.683  mm,	Y =   -143.940  mm,	Z =   -242.747  mm,
	W =  90.000 deg,	P =   0.000 deg,	R =   90.000 deg
};
P[756]{
   GP1:
	UF : 0, UT : 6,		CONFIG : 'N U T, 0, 0, 0',
	X =  316.886  mm,	Y =   -144.418  mm,	Z =   -242.790  mm,
	W =  90.000 deg,	P =   0.000 deg,	R =   90.000 deg
};
P[757]{
   GP1:
	UF : 0, UT : 6,		CONFIG : 'N U T, 0, 0, 0',
	X =  316.184  mm,	Y =   -144.771  mm,	Z =   -242.666  mm,
	W =  90.000 deg,	P =   0.000 deg,	R =   90.000 deg
};
P[758]{
   GP1:
	UF : 0, UT : 6,		CONFIG : 'N U T, 0, 0, 0',
	X =  313.977  mm,	Y =   -146.103  mm,	Z =   -242.804  mm,
	W =  90.000 deg,	P =   0.000 deg,	R =   90.000 deg
};
P[759]{
   GP1:
	UF : 0, UT : 6,		CONFIG : 'N U T, 0, 0, 0',
	X =  312.215  mm,	Y =   -147.070  mm,	Z =   -242.683  mm,
	W =  90.000 deg,	P =   0.000 deg,	R =   90.000 deg
};
P[760]{
   GP1:
	UF : 0, UT : 6,		CONFIG : 'N U T, 0, 0, 0',
	X =  309.541  mm,	Y =   -148.691  mm,	Z =   -242.868  mm,
	W =  90.000 deg,	P =   0.000 deg,	R =   90.000 deg
};
P[761]{
   GP1:
	UF : 0, UT : 6,		CONFIG : 'N U T, 0, 0, 0',
	X =  307.492  mm,	Y =   -149.911  mm,	Z =   -242.958  mm,
	W =  90.000 deg,	P =   0.000 deg,	R =   90.000 deg
};
P[762]{
   GP1:
	UF : 0, UT : 6,		CONFIG : 'N U T, 0, 0, 0',
	X =  304.198  mm,	Y =   -151.735  mm,	Z =   -242.769  mm,
	W =  90.000 deg,	P =   0.000 deg,	R =   90.000 deg
};
P[763]{
   GP1:
	UF : 0, UT : 6,		CONFIG : 'N U T, 0, 0, 0',
	X =  302.441  mm,	Y =   -152.745  mm,	Z =   -242.756  mm,
	W =  90.000 deg,	P =   0.000 deg,	R =   90.000 deg
};
P[764]{
   GP1:
	UF : 0, UT : 6,		CONFIG : 'N U T, 0, 0, 0',
	X =  301.538  mm,	Y =   -153.291  mm,	Z =   -242.816  mm,
	W =  90.000 deg,	P =   0.000 deg,	R =   90.000 deg
};
P[765]{
   GP1:
	UF : 0, UT : 6,		CONFIG : 'N U T, 0, 0, 0',
	X =  299.586  mm,	Y =   -154.450  mm,	Z =   -242.895  mm,
	W =  90.000 deg,	P =   0.000 deg,	R =   90.000 deg
};
P[766]{
   GP1:
	UF : 0, UT : 6,		CONFIG : 'N U T, 0, 0, 0',
	X =  298.582  mm,	Y =   -154.926  mm,	Z =   -242.646  mm,
	W =  90.000 deg,	P =   0.000 deg,	R =   90.000 deg
};
P[767]{
   GP1:
	UF : 0, UT : 6,		CONFIG : 'N U T, 0, 0, 0',
	X =  297.031  mm,	Y =   -155.899  mm,	Z =   -242.833  mm,
	W =  90.000 deg,	P =   0.000 deg,	R =   90.000 deg
};
P[768]{
   GP1:
	UF : 0, UT : 6,		CONFIG : 'N U T, 0, 0, 0',
	X =  290.958  mm,	Y =   -159.366  mm,	Z =   -242.734  mm,
	W =  90.000 deg,	P =   0.000 deg,	R =   90.000 deg
};
P[769]{
   GP1:
	UF : 0, UT : 6,		CONFIG : 'N U T, 0, 0, 0',
	X =  290.123  mm,	Y =   -160.011  mm,	Z =   -243.128  mm,
	W =  90.000 deg,	P =   0.000 deg,	R =   90.000 deg
};
P[770]{
   GP1:
	UF : 0, UT : 6,		CONFIG : 'N U T, 0, 0, 0',
	X =  287.276  mm,	Y =   -161.546  mm,	Z =   -242.867  mm,
	W =  90.000 deg,	P =   0.000 deg,	R =   90.000 deg
};
P[771]{
   GP1:
	UF : 0, UT : 6,		CONFIG : 'N U T, 0, 0, 0',
	X =  286.402  mm,	Y =   -161.977  mm,	Z =   -242.689  mm,
	W =  90.000 deg,	P =   0.000 deg,	R =   90.000 deg
};
P[772]{
   GP1:
	UF : 0, UT : 6,		CONFIG : 'N U T, 0, 0, 0',
	X =  284.847  mm,	Y =   -162.874  mm,	Z =   -242.687  mm,
	W =  90.000 deg,	P =   0.000 deg,	R =   90.000 deg
};
P[773]{
   GP1:
	UF : 0, UT : 6,		CONFIG : 'N U T, 0, 0, 0',
	X =  281.261  mm,	Y =   -165.073  mm,	Z =   -242.998  mm,
	W =  90.000 deg,	P =   0.000 deg,	R =   90.000 deg
};
P[774]{
   GP1:
	UF : 0, UT : 6,		CONFIG : 'N U T, 0, 0, 0',
	X =  279.845  mm,	Y =   -165.921  mm,	Z =   -243.073  mm,
	W =  90.000 deg,	P =   0.000 deg,	R =   90.000 deg
};
P[775]{
   GP1:
	UF : 0, UT : 6,		CONFIG : 'N U T, 0, 0, 0',
	X =  278.648  mm,	Y =   -166.490  mm,	Z =   -242.776  mm,
	W =  90.000 deg,	P =   0.000 deg,	R =   90.000 deg
};
P[776]{
   GP1:
	UF : 0, UT : 6,		CONFIG : 'N U T, 0, 0, 0',
	X =  276.497  mm,	Y =   -167.774  mm,	Z =   -242.879  mm,
	W =  90.000 deg,	P =   0.000 deg,	R =   90.000 deg
};
P[777]{
   GP1:
	UF : 0, UT : 6,		CONFIG : 'N U T, 0, 0, 0',
	X =  275.349  mm,	Y =   -168.363  mm,	Z =   -242.699  mm,
	W =  90.000 deg,	P =   0.000 deg,	R =   90.000 deg
};
P[778]{
   GP1:
	UF : 0, UT : 6,		CONFIG : 'N U T, 0, 0, 0',
	X =  273.717  mm,	Y =   -169.439  mm,	Z =   -243.021  mm,
	W =  90.000 deg,	P =   0.000 deg,	R =   90.000 deg
};
P[779]{
   GP1:
	UF : 0, UT : 6,		CONFIG : 'N U T, 0, 0, 0',
	X =  272.566  mm,	Y =   -170.031  mm,	Z =   -242.846  mm,
	W =  90.000 deg,	P =   0.000 deg,	R =   90.000 deg
};
P[780]{
   GP1:
	UF : 0, UT : 6,		CONFIG : 'N U T, 0, 0, 0',
	X =  271.866  mm,	Y =   -170.413  mm,	Z =   -242.793  mm,
	W =  90.000 deg,	P =   0.000 deg,	R =   90.000 deg
};
P[781]{
   GP1:
	UF : 0, UT : 6,		CONFIG : 'N U T, 0, 0, 0',
	X =  268.383  mm,	Y =   -172.496  mm,	Z =   -242.968  mm,
	W =  90.000 deg,	P =   0.000 deg,	R =   90.000 deg
};
P[782]{
   GP1:
	UF : 0, UT : 6,		CONFIG : 'N U T, 0, 0, 0',
	X =  266.155  mm,	Y =   -173.669  mm,	Z =   -242.691  mm,
	W =  90.000 deg,	P =   0.000 deg,	R =   90.000 deg
};
P[783]{
   GP1:
	UF : 0, UT : 6,		CONFIG : 'N U T, 0, 0, 0',
	X =  264.614  mm,	Y =   -174.653  mm,	Z =   -242.923  mm,
	W =  90.000 deg,	P =   0.000 deg,	R =   90.000 deg
};
P[784]{
   GP1:
	UF : 0, UT : 6,		CONFIG : 'N U T, 0, 0, 0',
	X =  263.441  mm,	Y =   -175.345  mm,	Z =   -242.955  mm,
	W =  90.000 deg,	P =   0.000 deg,	R =   90.000 deg
};
P[785]{
   GP1:
	UF : 0, UT : 6,		CONFIG : 'N U T, 0, 0, 0',
	X =  261.542  mm,	Y =   -176.312  mm,	Z =   -242.641  mm,
	W =  90.000 deg,	P =   0.000 deg,	R =   90.000 deg
};
P[786]{
   GP1:
	UF : 0, UT : 6,		CONFIG : 'N U T, 0, 0, 0',
	X =  258.287  mm,	Y =   -178.292  mm,	Z =   -242.886  mm,
	W =  90.000 deg,	P =   0.000 deg,	R =   90.000 deg
};
P[787]{
   GP1:
	UF : 0, UT : 6,		CONFIG : 'N U T, 0, 0, 0',
	X =  255.766  mm,	Y =   -179.651  mm,	Z =   -242.652  mm,
	W =  90.000 deg,	P =   0.000 deg,	R =   90.000 deg
};
P[788]{
   GP1:
	UF : 0, UT : 6,		CONFIG : 'N U T, 0, 0, 0',
	X =  254.355  mm,	Y =   -180.569  mm,	Z =   -242.903  mm,
	W =  90.000 deg,	P =   0.000 deg,	R =   90.000 deg
};
P[789]{
   GP1:
	UF : 0, UT : 6,		CONFIG : 'N U T, 0, 0, 0',
	X =  253.513  mm,	Y =   -180.954  mm,	Z =   -242.657  mm,
	W =  90.000 deg,	P =   0.000 deg,	R =   90.000 deg
};
P[790]{
   GP1:
	UF : 0, UT : 6,		CONFIG : 'N U T, 0, 0, 0',
	X =  252.948  mm,	Y =   -181.371  mm,	Z =   -242.879  mm,
	W =  90.000 deg,	P =   0.000 deg,	R =   90.000 deg
};
P[791]{
   GP1:
	UF : 0, UT : 6,		CONFIG : 'N U T, 0, 0, 0',
	X =  252.072  mm,	Y =   -181.876  mm,	Z =   -242.878  mm,
	W =  90.000 deg,	P =   0.000 deg,	R =   90.000 deg
};
P[792]{
   GP1:
	UF : 0, UT : 6,		CONFIG : 'N U T, 0, 0, 0',
	X =  249.867  mm,	Y =   -183.073  mm,	Z =   -242.690  mm,
	W =  90.000 deg,	P =   0.000 deg,	R =   90.000 deg
};
P[793]{
   GP1:
	UF : 0, UT : 6,		CONFIG : 'N U T, 0, 0, 0',
	X =  248.857  mm,	Y =   -183.649  mm,	Z =   -242.673  mm,
	W =  90.000 deg,	P =   0.000 deg,	R =   90.000 deg
};
P[794]{
   GP1:
	UF : 0, UT : 6,		CONFIG : 'N U T, 0, 0, 0',
	X =  247.939  mm,	Y =   -184.175  mm,	Z =   -242.665  mm,
	W =  90.000 deg,	P =   0.000 deg,	R =   90.000 deg
};
P[795]{
   GP1:
	UF : 0, UT : 6,		CONFIG : 'N U T, 0, 0, 0',
	X =  246.492  mm,	Y =   -185.026  mm,	Z =   -242.699  mm,
	W =  90.000 deg,	P =   0.000 deg,	R =   90.000 deg
};
P[796]{
   GP1:
	UF : 0, UT : 6,		CONFIG : 'N U T, 0, 0, 0',
	X =  244.448  mm,	Y =   -186.326  mm,	Z =   -242.992  mm,
	W =  90.000 deg,	P =   0.000 deg,	R =   90.000 deg
};
P[797]{
   GP1:
	UF : 0, UT : 6,		CONFIG : 'N U T, 0, 0, 0',
	X =  240.616  mm,	Y =   -188.545  mm,	Z =   -243.008  mm,
	W =  90.000 deg,	P =   0.000 deg,	R =   90.000 deg
};
P[798]{
   GP1:
	UF : 0, UT : 6,		CONFIG : 'N U T, 0, 0, 0',
	X =  238.228  mm,	Y =   -189.772  mm,	Z =   -242.640  mm,
	W =  90.000 deg,	P =   0.000 deg,	R =   90.000 deg
};
P[799]{
   GP1:
	UF : 0, UT : 6,		CONFIG : 'N U T, 0, 0, 0',
	X =  235.813  mm,	Y =   -191.212  mm,	Z =   -242.750  mm,
	W =  90.000 deg,	P =   0.000 deg,	R =   90.000 deg
};
P[800]{
   GP1:
	UF : 0, UT : 6,		CONFIG : 'N U T, 0, 0, 0',
	X =  234.762  mm,	Y =   -191.822  mm,	Z =   -242.757  mm,
	W =  90.000 deg,	P =   0.000 deg,	R =   90.000 deg
};
P[801]{
   GP1:
	UF : 0, UT : 6,		CONFIG : 'N U T, 0, 0, 0',
	X =  232.670  mm,	Y =   -193.011  mm,	Z =   -242.712  mm,
	W =  90.000 deg,	P =   0.000 deg,	R =   90.000 deg
};
P[802]{
   GP1:
	UF : 0, UT : 6,		CONFIG : 'N U T, 0, 0, 0',
	X =  232.075  mm,	Y =   -193.481  mm,	Z =   -243.020  mm,
	W =  90.000 deg,	P =   0.000 deg,	R =   90.000 deg
};
P[803]{
   GP1:
	UF : 0, UT : 6,		CONFIG : 'N U T, 0, 0, 0',
	X =  230.482  mm,	Y =   -194.275  mm,	Z =   -242.715  mm,
	W =  90.000 deg,	P =   0.000 deg,	R =   90.000 deg
};
P[804]{
   GP1:
	UF : 0, UT : 6,		CONFIG : 'N U T, 0, 0, 0',
	X =  230.167  mm,	Y =   -194.605  mm,	Z =   -243.074  mm,
	W =  90.000 deg,	P =   0.000 deg,	R =   90.000 deg
};
P[805]{
   GP1:
	UF : 0, UT : 6,		CONFIG : 'N U T, 0, 0, 0',
	X =  228.955  mm,	Y =   -195.225  mm,	Z =   -242.879  mm,
	W =  90.000 deg,	P =   0.000 deg,	R =   90.000 deg
};
P[806]{
   GP1:
	UF : 0, UT : 6,		CONFIG : 'N U T, 0, 0, 0',
	X =  228.304  mm,	Y =   -195.576  mm,	Z =   -242.819  mm,
	W =  90.000 deg,	P =   0.000 deg,	R =   90.000 deg
};
P[807]{
   GP1:
	UF : 0, UT : 6,		CONFIG : 'N U T, 0, 0, 0',
	X =  226.972  mm,	Y =   -196.373  mm,	Z =   -242.885  mm,
	W =  90.000 deg,	P =   0.000 deg,	R =   90.000 deg
};
P[808]{
   GP1:
	UF : 0, UT : 6,		CONFIG : 'N U T, 0, 0, 0',
	X =  225.997  mm,	Y =   -196.879  mm,	Z =   -242.748  mm,
	W =  90.000 deg,	P =   0.000 deg,	R =   90.000 deg
};
P[809]{
   GP1:
	UF : 0, UT : 6,		CONFIG : 'N U T, 0, 0, 0',
	X =  225.258  mm,	Y =   -197.424  mm,	Z =   -243.035  mm,
	W =  90.000 deg,	P =   0.000 deg,	R =   90.000 deg
};
P[810]{
   GP1:
	UF : 0, UT : 6,		CONFIG : 'N U T, 0, 0, 0',
	X =  222.737  mm,	Y =   -198.741  mm,	Z =   -242.700  mm,
	W =  90.000 deg,	P =   0.000 deg,	R =   90.000 deg
};
P[811]{
   GP1:
	UF : 0, UT : 6,		CONFIG : 'N U T, 0, 0, 0',
	X =  219.588  mm,	Y =   -200.617  mm,	Z =   -242.841  mm,
	W =  90.000 deg,	P =   0.000 deg,	R =   90.000 deg
};
P[812]{
   GP1:
	UF : 0, UT : 6,		CONFIG : 'N U T, 0, 0, 0',
	X =  215.509  mm,	Y =   -203.029  mm,	Z =   -242.978  mm,
	W =  90.000 deg,	P =   0.000 deg,	R =   90.000 deg
};
P[813]{
   GP1:
	UF : 0, UT : 6,		CONFIG : 'N U T, 0, 0, 0',
	X =  214.250  mm,	Y =   -203.745  mm,	Z =   -242.950  mm,
	W =  90.000 deg,	P =   0.000 deg,	R =   90.000 deg
};
P[814]{
   GP1:
	UF : 0, UT : 6,		CONFIG : 'N U T, 0, 0, 0',
	X =  213.030  mm,	Y =   -204.352  mm,	Z =   -242.714  mm,
	W =  90.000 deg,	P =   0.000 deg,	R =   90.000 deg
};
P[815]{
   GP1:
	UF : 0, UT : 6,		CONFIG : 'N U T, 0, 0, 0',
	X =  211.841  mm,	Y =   -205.058  mm,	Z =   -242.761  mm,
	W =  90.000 deg,	P =   0.000 deg,	R =   90.000 deg
};
P[816]{
   GP1:
	UF : 0, UT : 6,		CONFIG : 'N U T, 0, 0, 0',
	X =  211.045  mm,	Y =   -205.479  mm,	Z =   -242.668  mm,
	W =  90.000 deg,	P =   0.000 deg,	R =   90.000 deg
};
P[817]{
   GP1:
	UF : 0, UT : 6,		CONFIG : 'N U T, 0, 0, 0',
	X =  207.716  mm,	Y =   -207.439  mm,	Z =   -242.761  mm,
	W =  90.000 deg,	P =   0.000 deg,	R =   90.000 deg
};
P[818]{
   GP1:
	UF : 0, UT : 6,		CONFIG : 'N U T, 0, 0, 0',
	X =  206.550  mm,	Y =   -208.265  mm,	Z =   -243.131  mm,
	W =  90.000 deg,	P =   0.000 deg,	R =   90.000 deg
};
P[819]{
   GP1:
	UF : 0, UT : 6,		CONFIG : 'N U T, 0, 0, 0',
	X =  204.910  mm,	Y =   -209.121  mm,	Z =   -242.908  mm,
	W =  90.000 deg,	P =   0.000 deg,	R =   90.000 deg
};
P[820]{
   GP1:
	UF : 0, UT : 6,		CONFIG : 'N U T, 0, 0, 0',
	X =  203.677  mm,	Y =   -209.780  mm,	Z =   -242.781  mm,
	W =  90.000 deg,	P =   0.000 deg,	R =   90.000 deg
};
P[821]{
   GP1:
	UF : 0, UT : 6,		CONFIG : 'N U T, 0, 0, 0',
	X =  202.081  mm,	Y =   -210.841  mm,	Z =   -243.120  mm,
	W =  90.000 deg,	P =   0.000 deg,	R =   90.000 deg
};
P[822]{
   GP1:
	UF : 0, UT : 6,		CONFIG : 'N U T, 0, 0, 0',
	X =  199.930  mm,	Y =   -211.971  mm,	Z =   -242.848  mm,
	W =  90.000 deg,	P =   0.000 deg,	R =   90.000 deg
};
P[823]{
   GP1:
	UF : 0, UT : 6,		CONFIG : 'N U T, 0, 0, 0',
	X =  196.442  mm,	Y =   -214.064  mm,	Z =   -243.039  mm,
	W =  90.000 deg,	P =   0.000 deg,	R =   90.000 deg
};
P[824]{
   GP1:
	UF : 0, UT : 6,		CONFIG : 'N U T, 0, 0, 0',
	X =  195.768  mm,	Y =   -214.340  mm,	Z =   -242.765  mm,
	W =  90.000 deg,	P =   0.000 deg,	R =   90.000 deg
};
P[825]{
   GP1:
	UF : 0, UT : 6,		CONFIG : 'N U T, 0, 0, 0',
	X =  194.244  mm,	Y =   -215.279  mm,	Z =   -242.908  mm,
	W =  90.000 deg,	P =   0.000 deg,	R =   90.000 deg
};
P[826]{
   GP1:
	UF : 0, UT : 6,		CONFIG : 'N U T, 0, 0, 0',
	X =  193.374  mm,	Y =   -215.793  mm,	Z =   -242.937  mm,
	W =  90.000 deg,	P =   0.000 deg,	R =   90.000 deg
};
P[827]{
   GP1:
	UF : 0, UT : 6,		CONFIG : 'N U T, 0, 0, 0',
	X =  192.226  mm,	Y =   -216.335  mm,	Z =   -242.643  mm,
	W =  90.000 deg,	P =   0.000 deg,	R =   90.000 deg
};
P[828]{
   GP1:
	UF : 0, UT : 6,		CONFIG : 'N U T, 0, 0, 0',
	X =  191.250  mm,	Y =   -216.965  mm,	Z =   -242.804  mm,
	W =  90.000 deg,	P =   0.000 deg,	R =   90.000 deg
};
P[829]{
   GP1:
	UF : 0, UT : 6,		CONFIG : 'N U T, 0, 0, 0',
	X =  187.741  mm,	Y =   -219.123  mm,	Z =   -243.124  mm,
	W =  90.000 deg,	P =   0.000 deg,	R =   90.000 deg
};
P[830]{
   GP1:
	UF : 0, UT : 6,		CONFIG : 'N U T, 0, 0, 0',
	X =  186.411  mm,	Y =   -219.764  mm,	Z =   -242.816  mm,
	W =  90.000 deg,	P =   0.000 deg,	R =   90.000 deg
};
P[831]{
   GP1:
	UF : 0, UT : 6,		CONFIG : 'N U T, 0, 0, 0',
	X =  184.367  mm,	Y =   -220.960  mm,	Z =   -242.854  mm,
	W =  90.000 deg,	P =   0.000 deg,	R =   90.000 deg
};
P[832]{
   GP1:
	UF : 0, UT : 6,		CONFIG : 'N U T, 0, 0, 0',
	X =  182.485  mm,	Y =   -222.033  mm,	Z =   -242.823  mm,
	W =  90.000 deg,	P =   0.000 deg,	R =   90.000 deg
};
P[833]{
   GP1:
	UF : 0, UT : 6,		CONFIG : 'N U T, 0, 0, 0',
	X =  181.682  mm,	Y =   -222.524  mm,	Z =   -242.888  mm,
	W =  90.000 deg,	P =   0.000 deg,	R =   90.000 deg
};
P[834]{
   GP1:
	UF : 0, UT : 6,		CONFIG : 'N U T, 0, 0, 0',
	X =  180.651  mm,	Y =   -223.106  mm,	Z =   -242.857  mm,
	W =  90.000 deg,	P =   0.000 deg,	R =   90.000 deg
};
P[835]{
   GP1:
	UF : 0, UT : 6,		CONFIG : 'N U T, 0, 0, 0',
	X =  179.614  mm,	Y =   -223.627  mm,	Z =   -242.669  mm,
	W =  90.000 deg,	P =   0.000 deg,	R =   90.000 deg
};
P[836]{
   GP1:
	UF : 0, UT : 6,		CONFIG : 'N U T, 0, 0, 0',
	X =  176.615  mm,	Y =   -225.344  mm,	Z =   -242.633  mm,
	W =  90.000 deg,	P =   0.000 deg,	R =   90.000 deg
};
P[837]{
   GP1:
	UF : 0, UT : 6,		CONFIG : 'N U T, 0, 0, 0',
	X =  175.780  mm,	Y =   -225.912  mm,	Z =   -242.840  mm,
	W =  90.000 deg,	P =   0.000 deg,	R =   90.000 deg
};
P[838]{
   GP1:
	UF : 0, UT : 6,		CONFIG : 'N U T, 0, 0, 0',
	X =  173.477  mm,	Y =   -227.176  mm,	Z =   -242.682  mm,
	W =  90.000 deg,	P =   0.000 deg,	R =   90.000 deg
};
P[839]{
   GP1:
	UF : 0, UT : 6,		CONFIG : 'N U T, 0, 0, 0',
	X =  171.724  mm,	Y =   -228.174  mm,	Z =   -242.646  mm,
	W =  90.000 deg,	P =   0.000 deg,	R =   90.000 deg
};
P[840]{
   GP1:
	UF : 0, UT : 6,		CONFIG : 'N U T, 0, 0, 0',
	X =  166.240  mm,	Y =   -231.492  mm,	Z =   -243.015  mm,
	W =  90.000 deg,	P =   0.000 deg,	R =   90.000 deg
};
P[841]{
   GP1:
	UF : 0, UT : 6,		CONFIG : 'N U T, 0, 0, 0',
	X =  163.812  mm,	Y =   -232.820  mm,	Z =   -242.833  mm,
	W =  90.000 deg,	P =   0.000 deg,	R =   90.000 deg
};
P[842]{
   GP1:
	UF : 0, UT : 6,		CONFIG : 'N U T, 0, 0, 0',
	X =  159.100  mm,	Y =   -235.466  mm,	Z =   -242.654  mm,
	W =  90.000 deg,	P =   0.000 deg,	R =   90.000 deg
};
P[843]{
   GP1:
	UF : 0, UT : 6,		CONFIG : 'N U T, 0, 0, 0',
	X =  158.456  mm,	Y =   -235.851  mm,	Z =   -242.686  mm,
	W =  90.000 deg,	P =   0.000 deg,	R =   90.000 deg
};
P[844]{
   GP1:
	UF : 0, UT : 6,		CONFIG : 'N U T, 0, 0, 0',
	X =  157.551  mm,	Y =   -236.391  mm,	Z =   -242.729  mm,
	W =  90.000 deg,	P =   0.000 deg,	R =   90.000 deg
};
P[845]{
   GP1:
	UF : 0, UT : 6,		CONFIG : 'N U T, 0, 0, 0',
	X =  156.515  mm,	Y =   -237.066  mm,	Z =   -242.914  mm,
	W =  90.000 deg,	P =   0.000 deg,	R =   90.000 deg
};
P[846]{
   GP1:
	UF : 0, UT : 6,		CONFIG : 'N U T, 0, 0, 0',
	X =  155.042  mm,	Y =   -237.812  mm,	Z =   -242.660  mm,
	W =  90.000 deg,	P =   0.000 deg,	R =   90.000 deg
};
P[847]{
   GP1:
	UF : 0, UT : 6,		CONFIG : 'N U T, 0, 0, 0',
	X =  154.391  mm,	Y =   -238.307  mm,	Z =   -242.950  mm,
	W =  90.000 deg,	P =   0.000 deg,	R =   90.000 deg
};
P[848]{
   GP1:
	UF : 0, UT : 6,		CONFIG : 'N U T, 0, 0, 0',
	X =  153.655  mm,	Y =   -238.790  mm,	Z =   -243.091  mm,
	W =  90.000 deg,	P =   0.000 deg,	R =   90.000 deg
};
P[849]{
   GP1:
	UF : 0, UT : 6,		CONFIG : 'N U T, 0, 0, 0',
	X =  152.861  mm,	Y =   -239.129  mm,	Z =   -242.801  mm,
	W =  90.000 deg,	P =   0.000 deg,	R =   90.000 deg
};
P[850]{
   GP1:
	UF : 0, UT : 6,		CONFIG : 'N U T, 0, 0, 0',
	X =  150.970  mm,	Y =   -240.351  mm,	Z =   -243.117  mm,
	W =  90.000 deg,	P =   0.000 deg,	R =   90.000 deg
};
P[851]{
   GP1:
	UF : 0, UT : 6,		CONFIG : 'N U T, 0, 0, 0',
	X =  150.294  mm,	Y =   -240.596  mm,	Z =   -242.765  mm,
	W =  90.000 deg,	P =   0.000 deg,	R =   90.000 deg
};
P[852]{
   GP1:
	UF : 0, UT : 6,		CONFIG : 'N U T, 0, 0, 0',
	X =  149.104  mm,	Y =   -241.245  mm,	Z =   -242.673  mm,
	W =  90.000 deg,	P =   0.000 deg,	R =   90.000 deg
};
P[853]{
   GP1:
	UF : 0, UT : 6,		CONFIG : 'N U T, 0, 0, 0',
	X =  148.113  mm,	Y =   -242.002  mm,	Z =   -243.123  mm,
	W =  90.000 deg,	P =   0.000 deg,	R =   90.000 deg
};
P[854]{
   GP1:
	UF : 0, UT : 6,		CONFIG : 'N U T, 0, 0, 0',
	X =  147.507  mm,	Y =   -242.236  mm,	Z =   -242.840  mm,
	W =  90.000 deg,	P =   0.000 deg,	R =   90.000 deg
};
P[855]{
   GP1:
	UF : 0, UT : 6,		CONFIG : 'N U T, 0, 0, 0',
	X =  144.089  mm,	Y =   -244.322  mm,	Z =   -243.112  mm,
	W =  90.000 deg,	P =   0.000 deg,	R =   90.000 deg
};
P[856]{
   GP1:
	UF : 0, UT : 6,		CONFIG : 'N U T, 0, 0, 0',
	X =  139.773  mm,	Y =   -246.676  mm,	Z =   -242.777  mm,
	W =  90.000 deg,	P =   0.000 deg,	R =   90.000 deg
};
P[857]{
   GP1:
	UF : 0, UT : 6,		CONFIG : 'N U T, 0, 0, 0',
	X =  138.576  mm,	Y =   -247.380  mm,	Z =   -242.808  mm,
	W =  90.000 deg,	P =   0.000 deg,	R =   90.000 deg
};
P[858]{
   GP1:
	UF : 0, UT : 6,		CONFIG : 'N U T, 0, 0, 0',
	X =  136.940  mm,	Y =   -248.406  mm,	Z =   -243.008  mm,
	W =  90.000 deg,	P =   0.000 deg,	R =   90.000 deg
};
P[859]{
   GP1:
	UF : 0, UT : 6,		CONFIG : 'N U T, 0, 0, 0',
	X =  136.197  mm,	Y =   -248.739  mm,	Z =   -242.773  mm,
	W =  90.000 deg,	P =   0.000 deg,	R =   90.000 deg
};
P[860]{
   GP1:
	UF : 0, UT : 6,		CONFIG : 'N U T, 0, 0, 0',
	X =  135.217  mm,	Y =   -249.409  mm,	Z =   -243.025  mm,
	W =  90.000 deg,	P =   0.000 deg,	R =   90.000 deg
};
P[861]{
   GP1:
	UF : 0, UT : 6,		CONFIG : 'N U T, 0, 0, 0',
	X =  132.593  mm,	Y =   -250.924  mm,	Z =   -243.024  mm,
	W =  90.000 deg,	P =   0.000 deg,	R =   90.000 deg
};
P[862]{
   GP1:
	UF : 0, UT : 6,		CONFIG : 'N U T, 0, 0, 0',
	X =  131.674  mm,	Y =   -251.399  mm,	Z =   -242.890  mm,
	W =  90.000 deg,	P =   0.000 deg,	R =   90.000 deg
};
P[863]{
   GP1:
	UF : 0, UT : 6,		CONFIG : 'N U T, 0, 0, 0',
	X =  130.976  mm,	Y =   -251.716  mm,	Z =   -242.681  mm,
	W =  90.000 deg,	P =   0.000 deg,	R =   90.000 deg
};
P[864]{
   GP1:
	UF : 0, UT : 6,		CONFIG : 'N U T, 0, 0, 0',
	X =  129.281  mm,	Y =   -252.838  mm,	Z =   -243.030  mm,
	W =  90.000 deg,	P =   0.000 deg,	R =   90.000 deg
};
P[865]{
   GP1:
	UF : 0, UT : 6,		CONFIG : 'N U T, 0, 0, 0',
	X =  128.500  mm,	Y =   -253.187  mm,	Z =   -242.782  mm,
	W =  90.000 deg,	P =   0.000 deg,	R =   90.000 deg
};
P[866]{
   GP1:
	UF : 0, UT : 6,		CONFIG : 'N U T, 0, 0, 0',
	X =  127.830  mm,	Y =   -253.575  mm,	Z =   -242.787  mm,
	W =  90.000 deg,	P =   0.000 deg,	R =   90.000 deg
};
P[867]{
   GP1:
	UF : 0, UT : 6,		CONFIG : 'N U T, 0, 0, 0',
	X =  126.858  mm,	Y =   -254.115  mm,	Z =   -242.733  mm,
	W =  90.000 deg,	P =   0.000 deg,	R =   90.000 deg
};
P[868]{
   GP1:
	UF : 0, UT : 6,		CONFIG : 'N U T, 0, 0, 0',
	X =  125.184  mm,	Y =   -255.199  mm,	Z =   -243.020  mm,
	W =  90.000 deg,	P =   0.000 deg,	R =   90.000 deg
};
P[869]{
   GP1:
	UF : 0, UT : 6,		CONFIG : 'N U T, 0, 0, 0',
	X =  122.790  mm,	Y =   -256.502  mm,	Z =   -242.828  mm,
	W =  90.000 deg,	P =   0.000 deg,	R =   90.000 deg
};
P[870]{
   GP1:
	UF : 0, UT : 6,		CONFIG : 'N U T, 0, 0, 0',
	X =  121.786  mm,	Y =   -257.044  mm,	Z =   -242.735  mm,
	W =  90.000 deg,	P =   0.000 deg,	R =   90.000 deg
};
P[871]{
   GP1:
	UF : 0, UT : 6,		CONFIG : 'N U T, 0, 0, 0',
	X =  119.886  mm,	Y =   -258.199  mm,	Z =   -242.875  mm,
	W =  90.000 deg,	P =   0.000 deg,	R =   90.000 deg
};
P[872]{
   GP1:
	UF : 0, UT : 6,		CONFIG : 'N U T, 0, 0, 0',
	X =  118.487  mm,	Y =   -258.949  mm,	Z =   -242.733  mm,
	W =  90.000 deg,	P =   0.000 deg,	R =   90.000 deg
};
P[873]{
   GP1:
	UF : 0, UT : 6,		CONFIG : 'N U T, 0, 0, 0',
	X =  116.860  mm,	Y =   -260.000  mm,	Z =   -243.006  mm,
	W =  90.000 deg,	P =   0.000 deg,	R =   90.000 deg
};
P[874]{
   GP1:
	UF : 0, UT : 6,		CONFIG : 'N U T, 0, 0, 0',
	X =  115.708  mm,	Y =   -260.575  mm,	Z =   -242.789  mm,
	W =  90.000 deg,	P =   0.000 deg,	R =   90.000 deg
};
P[875]{
   GP1:
	UF : 0, UT : 6,		CONFIG : 'N U T, 0, 0, 0',
	X =  115.089  mm,	Y =   -260.946  mm,	Z =   -242.823  mm,
	W =  90.000 deg,	P =   0.000 deg,	R =   90.000 deg
};
P[876]{
   GP1:
	UF : 0, UT : 6,		CONFIG : 'N U T, 0, 0, 0',
	X =  113.757  mm,	Y =   -261.834  mm,	Z =   -243.110  mm,
	W =  90.000 deg,	P =   0.000 deg,	R =   90.000 deg
};
P[877]{
   GP1:
	UF : 0, UT : 6,		CONFIG : 'N U T, 0, 0, 0',
	X =  111.802  mm,	Y =   -262.963  mm,	Z =   -243.109  mm,
	W =  90.000 deg,	P =   0.000 deg,	R =   90.000 deg
};
P[878]{
   GP1:
	UF : 0, UT : 6,		CONFIG : 'N U T, 0, 0, 0',
	X =  110.830  mm,	Y =   -263.371  mm,	Z =   -242.736  mm,
	W =  90.000 deg,	P =   0.000 deg,	R =   90.000 deg
};
P[879]{
   GP1:
	UF : 0, UT : 6,		CONFIG : 'N U T, 0, 0, 0',
	X =  107.379  mm,	Y =   -262.614  mm,	Z =   -236.061  mm,
	W =  90.000 deg,	P =   0.000 deg,	R =   90.000 deg
};
P[880]{
   GP1:
	UF : 0, UT : 6,		CONFIG : 'N U T, 0, 0, 0',
	X =  106.362  mm,	Y =   -263.194  mm,	Z =   -236.046  mm,
	W =  90.000 deg,	P =   0.000 deg,	R =   90.000 deg
};
P[881]{
   GP1:
	UF : 0, UT : 6,		CONFIG : 'N U T, 0, 0, 0',
	X =  102.626  mm,	Y =   -265.397  mm,	Z =   -236.158  mm,
	W =  90.000 deg,	P =   0.000 deg,	R =   90.000 deg
};
P[882]{
   GP1:
	UF : 0, UT : 6,		CONFIG : 'N U T, 0, 0, 0',
	X =  101.694  mm,	Y =   -265.781  mm,	Z =   -235.782  mm,
	W =  90.000 deg,	P =   0.000 deg,	R =   90.000 deg
};
P[883]{
   GP1:
	UF : 0, UT : 6,		CONFIG : 'N U T, 0, 0, 0',
	X =  101.244  mm,	Y =   -266.178  mm,	Z =   -236.117  mm,
	W =  90.000 deg,	P =   0.000 deg,	R =   90.000 deg
};
P[884]{
   GP1:
	UF : 0, UT : 6,		CONFIG : 'N U T, 0, 0, 0',
	X =  99.521  mm,	Y =   -267.225  mm,	Z =   -236.242  mm,
	W =  90.000 deg,	P =   0.000 deg,	R =   90.000 deg
};
P[885]{
   GP1:
	UF : 0, UT : 6,		CONFIG : 'N U T, 0, 0, 0',
	X =  97.714  mm,	Y =   -268.266  mm,	Z =   -236.238  mm,
	W =  90.000 deg,	P =   0.000 deg,	R =   90.000 deg
};
P[886]{
   GP1:
	UF : 0, UT : 6,		CONFIG : 'N U T, 0, 0, 0',
	X =  96.236  mm,	Y =   -268.955  mm,	Z =   -235.839  mm,
	W =  90.000 deg,	P =   0.000 deg,	R =   90.000 deg
};
P[887]{
   GP1:
	UF : 0, UT : 6,		CONFIG : 'N U T, 0, 0, 0',
	X =  95.700  mm,	Y =   -269.341  mm,	Z =   -236.024  mm,
	W =  90.000 deg,	P =   0.000 deg,	R =   90.000 deg
};
P[888]{
   GP1:
	UF : 0, UT : 6,		CONFIG : 'N U T, 0, 0, 0',
	X =  91.513  mm,	Y =   -271.810  mm,	Z =   -236.149  mm,
	W =  90.000 deg,	P =   0.000 deg,	R =   90.000 deg
};
P[889]{
   GP1:
	UF : 0, UT : 6,		CONFIG : 'N U T, 0, 0, 0',
	X =  88.409  mm,	Y =   -273.504  mm,	Z =   -235.912  mm,
	W =  90.000 deg,	P =   0.000 deg,	R =   90.000 deg
};
P[890]{
   GP1:
	UF : 0, UT : 6,		CONFIG : 'N U T, 0, 0, 0',
	X =  87.323  mm,	Y =   -274.228  mm,	Z =   -236.147  mm,
	W =  90.000 deg,	P =   0.000 deg,	R =   90.000 deg
};
P[891]{
   GP1:
	UF : 0, UT : 6,		CONFIG : 'N U T, 0, 0, 0',
	X =  84.978  mm,	Y =   -275.573  mm,	Z =   -236.124  mm,
	W =  90.000 deg,	P =   0.000 deg,	R =   90.000 deg
};
P[892]{
   GP1:
	UF : 0, UT : 6,		CONFIG : 'N U T, 0, 0, 0',
	X =  84.347  mm,	Y =   -275.980  mm,	Z =   -236.226  mm,
	W =  90.000 deg,	P =   0.000 deg,	R =   90.000 deg
};
P[893]{
   GP1:
	UF : 0, UT : 6,		CONFIG : 'N U T, 0, 0, 0',
	X =  83.616  mm,	Y =   -276.378  mm,	Z =   -236.169  mm,
	W =  90.000 deg,	P =   0.000 deg,	R =   90.000 deg
};
P[894]{
   GP1:
	UF : 0, UT : 6,		CONFIG : 'N U T, 0, 0, 0',
	X =  81.161  mm,	Y =   -277.777  mm,	Z =   -236.125  mm,
	W =  90.000 deg,	P =   0.000 deg,	R =   90.000 deg
};
P[895]{
   GP1:
	UF : 0, UT : 6,		CONFIG : 'N U T, 0, 0, 0',
	X =  80.172  mm,	Y =   -278.254  mm,	Z =   -235.896  mm,
	W =  90.000 deg,	P =   0.000 deg,	R =   90.000 deg
};
P[896]{
   GP1:
	UF : 0, UT : 6,		CONFIG : 'N U T, 0, 0, 0',
	X =  77.773  mm,	Y =   -279.776  mm,	Z =   -236.230  mm,
	W =  90.000 deg,	P =   0.000 deg,	R =   90.000 deg
};
P[897]{
   GP1:
	UF : 0, UT : 6,		CONFIG : 'N U T, 0, 0, 0',
	X =  73.440  mm,	Y =   -282.290  mm,	Z =   -236.257  mm,
	W =  90.000 deg,	P =   0.000 deg,	R =   90.000 deg
};
P[898]{
   GP1:
	UF : 0, UT : 6,		CONFIG : 'N U T, 0, 0, 0',
	X =  70.388  mm,	Y =   -283.892  mm,	Z =   -235.869  mm,
	W =  90.000 deg,	P =   0.000 deg,	R =   90.000 deg
};
P[899]{
   GP1:
	UF : 0, UT : 6,		CONFIG : 'N U T, 0, 0, 0',
	X =  65.030  mm,	Y =   -287.146  mm,	Z =   -236.258  mm,
	W =  90.000 deg,	P =   0.000 deg,	R =   90.000 deg
};
P[900]{
   GP1:
	UF : 0, UT : 6,		CONFIG : 'N U T, 0, 0, 0',
	X =  63.436  mm,	Y =   -288.039  mm,	Z =   -236.191  mm,
	W =  90.000 deg,	P =   0.000 deg,	R =   90.000 deg
};
P[901]{
   GP1:
	UF : 0, UT : 6,		CONFIG : 'N U T, 0, 0, 0',
	X =  58.049  mm,	Y =   -291.156  mm,	Z =   -236.208  mm,
	W =  90.000 deg,	P =   0.000 deg,	R =   90.000 deg
};
P[902]{
   GP1:
	UF : 0, UT : 6,		CONFIG : 'N U T, 0, 0, 0',
	X =  57.340  mm,	Y =   -291.579  mm,	Z =   -236.242  mm,
	W =  90.000 deg,	P =   0.000 deg,	R =   90.000 deg
};
P[903]{
   GP1:
	UF : 0, UT : 6,		CONFIG : 'N U T, 0, 0, 0',
	X =  56.659  mm,	Y =   -291.781  mm,	Z =   -235.776  mm,
	W =  90.000 deg,	P =   0.000 deg,	R =   90.000 deg
};
P[904]{
   GP1:
	UF : 0, UT : 6,		CONFIG : 'N U T, 0, 0, 0',
	X =  55.700  mm,	Y =   -292.486  mm,	Z =   -236.144  mm,
	W =  90.000 deg,	P =   0.000 deg,	R =   90.000 deg
};
P[905]{
   GP1:
	UF : 0, UT : 6,		CONFIG : 'N U T, 0, 0, 0',
	X =  53.441  mm,	Y =   -293.824  mm,	Z =   -236.227  mm,
	W =  90.000 deg,	P =   0.000 deg,	R =   90.000 deg
};
P[906]{
   GP1:
	UF : 0, UT : 6,		CONFIG : 'N U T, 0, 0, 0',
	X =  52.670  mm,	Y =   -294.281  mm,	Z =   -236.255  mm,
	W =  90.000 deg,	P =   0.000 deg,	R =   90.000 deg
};
P[907]{
   GP1:
	UF : 0, UT : 6,		CONFIG : 'N U T, 0, 0, 0',
	X =  50.879  mm,	Y =   -295.214  mm,	Z =   -236.009  mm,
	W =  90.000 deg,	P =   0.000 deg,	R =   90.000 deg
};
P[908]{
   GP1:
	UF : 0, UT : 6,		CONFIG : 'N U T, 0, 0, 0',
	X =  50.144  mm,	Y =   -295.650  mm,	Z =   -236.036  mm,
	W =  90.000 deg,	P =   0.000 deg,	R =   90.000 deg
};
P[909]{
   GP1:
	UF : 0, UT : 6,		CONFIG : 'N U T, 0, 0, 0',
	X =  48.422  mm,	Y =   -296.721  mm,	Z =   -236.223  mm,
	W =  90.000 deg,	P =   0.000 deg,	R =   90.000 deg
};
P[910]{
   GP1:
	UF : 0, UT : 6,		CONFIG : 'N U T, 0, 0, 0',
	X =  46.970  mm,	Y =   -297.556  mm,	Z =   -236.217  mm,
	W =  90.000 deg,	P =   0.000 deg,	R =   90.000 deg
};
P[911]{
   GP1:
	UF : 0, UT : 6,		CONFIG : 'N U T, 0, 0, 0',
	X =  45.499  mm,	Y =   -298.257  mm,	Z =   -235.853  mm,
	W =  90.000 deg,	P =   0.000 deg,	R =   90.000 deg
};
P[912]{
   GP1:
	UF : 0, UT : 6,		CONFIG : 'N U T, 0, 0, 0',
	X =  44.834  mm,	Y =   -298.743  mm,	Z =   -236.104  mm,
	W =  90.000 deg,	P =   0.000 deg,	R =   90.000 deg
};
P[913]{
   GP1:
	UF : 0, UT : 6,		CONFIG : 'N U T, 0, 0, 0',
	X =  43.982  mm,	Y =   -299.129  mm,	Z =   -235.848  mm,
	W =  90.000 deg,	P =   0.000 deg,	R =   90.000 deg
};
P[914]{
   GP1:
	UF : 0, UT : 6,		CONFIG : 'N U T, 0, 0, 0',
	X =  42.850  mm,	Y =   -299.905  mm,	Z =   -236.142  mm,
	W =  90.000 deg,	P =   0.000 deg,	R =   90.000 deg
};
P[915]{
   GP1:
	UF : 0, UT : 6,		CONFIG : 'N U T, 0, 0, 0',
	X =  41.970  mm,	Y =   -300.345  mm,	Z =   -235.979  mm,
	W =  90.000 deg,	P =   0.000 deg,	R =   90.000 deg
};
P[916]{
   GP1:
	UF : 0, UT : 6,		CONFIG : 'N U T, 0, 0, 0',
	X =  39.796  mm,	Y =   -301.665  mm,	Z =   -236.133  mm,
	W =  90.000 deg,	P =   0.000 deg,	R =   90.000 deg
};
P[917]{
   GP1:
	UF : 0, UT : 6,		CONFIG : 'N U T, 0, 0, 0',
	X =  39.173  mm,	Y =   -302.056  mm,	Z =   -236.210  mm,
	W =  90.000 deg,	P =   0.000 deg,	R =   90.000 deg
};
P[918]{
   GP1:
	UF : 0, UT : 6,		CONFIG : 'N U T, 0, 0, 0',
	X =  38.479  mm,	Y =   -302.462  mm,	Z =   -236.224  mm,
	W =  90.000 deg,	P =   0.000 deg,	R =   90.000 deg
};
P[919]{
   GP1:
	UF : 0, UT : 6,		CONFIG : 'N U T, 0, 0, 0',
	X =  37.678  mm,	Y =   -302.927  mm,	Z =   -236.231  mm,
	W =  90.000 deg,	P =   0.000 deg,	R =   90.000 deg
};
P[920]{
   GP1:
	UF : 0, UT : 6,		CONFIG : 'N U T, 0, 0, 0',
	X =  36.185  mm,	Y =   -303.744  mm,	Z =   -236.121  mm,
	W =  90.000 deg,	P =   0.000 deg,	R =   90.000 deg
};
P[921]{
   GP1:
	UF : 0, UT : 6,		CONFIG : 'N U T, 0, 0, 0',
	X =  35.028  mm,	Y =   -304.448  mm,	Z =   -236.207  mm,
	W =  90.000 deg,	P =   0.000 deg,	R =   90.000 deg
};
P[922]{
   GP1:
	UF : 0, UT : 6,		CONFIG : 'N U T, 0, 0, 0',
	X =  34.079  mm,	Y =   -304.950  mm,	Z =   -236.097  mm,
	W =  90.000 deg,	P =   0.000 deg,	R =   90.000 deg
};
P[923]{
   GP1:
	UF : 0, UT : 6,		CONFIG : 'N U T, 0, 0, 0',
	X =  32.668  mm,	Y =   -305.794  mm,	Z =   -236.167  mm,
	W =  90.000 deg,	P =   0.000 deg,	R =   90.000 deg
};
P[924]{
   GP1:
	UF : 0, UT : 6,		CONFIG : 'N U T, 0, 0, 0',
	X =  31.971  mm,	Y =   -306.207  mm,	Z =   -236.193  mm,
	W =  90.000 deg,	P =   0.000 deg,	R =   90.000 deg
};
P[925]{
   GP1:
	UF : 0, UT : 6,		CONFIG : 'N U T, 0, 0, 0',
	X =  31.055  mm,	Y =   -306.696  mm,	Z =   -236.096  mm,
	W =  90.000 deg,	P =   0.000 deg,	R =   90.000 deg
};
P[926]{
   GP1:
	UF : 0, UT : 6,		CONFIG : 'N U T, 0, 0, 0',
	X =  29.602  mm,	Y =   -307.512  mm,	Z =   -236.043  mm,
	W =  90.000 deg,	P =   0.000 deg,	R =   90.000 deg
};
P[927]{
   GP1:
	UF : 0, UT : 6,		CONFIG : 'N U T, 0, 0, 0',
	X =  28.648  mm,	Y =   -308.151  mm,	Z =   -236.255  mm,
	W =  90.000 deg,	P =   0.000 deg,	R =   90.000 deg
};
P[928]{
   GP1:
	UF : 0, UT : 6,		CONFIG : 'N U T, 0, 0, 0',
	X =  27.827  mm,	Y =   -308.542  mm,	Z =   -236.052  mm,
	W =  90.000 deg,	P =   0.000 deg,	R =   90.000 deg
};
P[929]{
   GP1:
	UF : 0, UT : 6,		CONFIG : 'N U T, 0, 0, 0',
	X =  25.069  mm,	Y =   -310.092  mm,	Z =   -235.949  mm,
	W =  90.000 deg,	P =   0.000 deg,	R =   90.000 deg
};
P[930]{
   GP1:
	UF : 0, UT : 6,		CONFIG : 'N U T, 0, 0, 0',
	X =  23.271  mm,	Y =   -311.209  mm,	Z =   -236.143  mm,
	W =  90.000 deg,	P =   0.000 deg,	R =   90.000 deg
};
P[931]{
   GP1:
	UF : 0, UT : 6,		CONFIG : 'N U T, 0, 0, 0',
	X =  21.992  mm,	Y =   -311.957  mm,	Z =   -236.165  mm,
	W =  90.000 deg,	P =   0.000 deg,	R =   90.000 deg
};
P[932]{
   GP1:
	UF : 0, UT : 6,		CONFIG : 'N U T, 0, 0, 0',
	X =  18.458  mm,	Y =   -313.974  mm,	Z =   -236.108  mm,
	W =  90.000 deg,	P =   0.000 deg,	R =   90.000 deg
};
P[933]{
   GP1:
	UF : 0, UT : 6,		CONFIG : 'N U T, 0, 0, 0',
	X =  16.832  mm,	Y =   -314.947  mm,	Z =   -236.191  mm,
	W =  90.000 deg,	P =   0.000 deg,	R =   90.000 deg
};
P[934]{
   GP1:
	UF : 0, UT : 6,		CONFIG : 'N U T, 0, 0, 0',
	X =  15.396  mm,	Y =   -315.622  mm,	Z =   -235.816  mm,
	W =  90.000 deg,	P =   0.000 deg,	R =   90.000 deg
};
P[935]{
   GP1:
	UF : 0, UT : 6,		CONFIG : 'N U T, 0, 0, 0',
	X =  13.529  mm,	Y =   -316.865  mm,	Z =   -236.216  mm,
	W =  90.000 deg,	P =   0.000 deg,	R =   90.000 deg
};
P[936]{
   GP1:
	UF : 0, UT : 6,		CONFIG : 'N U T, 0, 0, 0',
	X =  10.124  mm,	Y =   -318.719  mm,	Z =   -235.945  mm,
	W =  90.000 deg,	P =   0.000 deg,	R =   90.000 deg
};
P[937]{
   GP1:
	UF : 0, UT : 6,		CONFIG : 'N U T, 0, 0, 0',
	X =  5.035  mm,	Y =   -321.742  mm,	Z =   -236.150  mm,
	W =  90.000 deg,	P =   0.000 deg,	R =   90.000 deg
};
P[938]{
   GP1:
	UF : 0, UT : 6,		CONFIG : 'N U T, 0, 0, 0',
	X =  3.379  mm,	Y =   -322.674  mm,	Z =   -236.091  mm,
	W =  90.000 deg,	P =   0.000 deg,	R =   90.000 deg
};
P[939]{
   GP1:
	UF : 0, UT : 6,		CONFIG : 'N U T, 0, 0, 0',
	X =  2.456  mm,	Y =   -323.209  mm,	Z =   -236.095  mm,
	W =  90.000 deg,	P =   0.000 deg,	R =   90.000 deg
};
P[940]{
   GP1:
	UF : 0, UT : 6,		CONFIG : 'N U T, 0, 0, 0',
	X =  0.779  mm,	Y =   -324.224  mm,	Z =   -236.211  mm,
	W =  90.000 deg,	P =   0.000 deg,	R =   90.000 deg
};
P[941]{
   GP1:
	UF : 0, UT : 6,		CONFIG : 'N U T, 0, 0, 0',
	X =  0.092  mm,	Y =   -324.593  mm,	Z =   -236.142  mm,
	W =  90.000 deg,	P =   0.000 deg,	R =   90.000 deg
};
P[942]{
   GP1:
	UF : 0, UT : 6,		CONFIG : 'N U T, 0, 0, 0',
	X =  -2.016  mm,	Y =   -325.780  mm,	Z =   -236.069  mm,
	W =  90.000 deg,	P =   0.000 deg,	R =   90.000 deg
};
P[943]{
   GP1:
	UF : 0, UT : 6,		CONFIG : 'N U T, 0, 0, 0',
	X =  -3.613  mm,	Y =   -326.649  mm,	Z =   -235.943  mm,
	W =  90.000 deg,	P =   0.000 deg,	R =   90.000 deg
};
P[944]{
   GP1:
	UF : 0, UT : 6,		CONFIG : 'N U T, 0, 0, 0',
	X =  -6.998  mm,	Y =   -328.558  mm,	Z =   -235.829  mm,
	W =  90.000 deg,	P =   0.000 deg,	R =   90.000 deg
};
P[945]{
   GP1:
	UF : 0, UT : 6,		CONFIG : 'N U T, 0, 0, 0',
	X =  -9.233  mm,	Y =   -330.012  mm,	Z =   -236.226  mm,
	W =  90.000 deg,	P =   0.000 deg,	R =   90.000 deg
};
P[946]{
   GP1:
	UF : 0, UT : 6,		CONFIG : 'N U T, 0, 0, 0',
	X =  -9.754  mm,	Y =   -330.241  mm,	Z =   -236.053  mm,
	W =  90.000 deg,	P =   0.000 deg,	R =   90.000 deg
};
P[947]{
   GP1:
	UF : 0, UT : 6,		CONFIG : 'N U T, 0, 0, 0',
	X =  -14.100  mm,	Y =   -332.825  mm,	Z =   -236.235  mm,
	W =  90.000 deg,	P =   0.000 deg,	R =   90.000 deg
};
P[948]{
   GP1:
	UF : 0, UT : 6,		CONFIG : 'N U T, 0, 0, 0',
	X =  -15.681  mm,	Y =   -333.619  mm,	Z =   -235.945  mm,
	W =  90.000 deg,	P =   0.000 deg,	R =   90.000 deg
};
P[949]{
   GP1:
	UF : 0, UT : 6,		CONFIG : 'N U T, 0, 0, 0',
	X =  -17.955  mm,	Y =   -335.032  mm,	Z =   -236.187  mm,
	W =  90.000 deg,	P =   0.000 deg,	R =   90.000 deg
};
P[950]{
   GP1:
	UF : 0, UT : 6,		CONFIG : 'N U T, 0, 0, 0',
	X =  -19.063  mm,	Y =   -335.617  mm,	Z =   -236.056  mm,
	W =  90.000 deg,	P =   0.000 deg,	R =   90.000 deg
};
P[951]{
   GP1:
	UF : 0, UT : 6,		CONFIG : 'N U T, 0, 0, 0',
	X =  -20.134  mm,	Y =   -336.315  mm,	Z =   -236.248  mm,
	W =  90.000 deg,	P =   0.000 deg,	R =   90.000 deg
};
P[952]{
   GP1:
	UF : 0, UT : 6,		CONFIG : 'N U T, 0, 0, 0',
	X =  -22.063  mm,	Y =   -337.351  mm,	Z =   -236.060  mm,
	W =  90.000 deg,	P =   0.000 deg,	R =   90.000 deg
};
P[953]{
   GP1:
	UF : 0, UT : 6,		CONFIG : 'N U T, 0, 0, 0',
	X =  -23.040  mm,	Y =   -337.861  mm,	Z =   -235.930  mm,
	W =  90.000 deg,	P =   0.000 deg,	R =   90.000 deg
};
P[954]{
   GP1:
	UF : 0, UT : 6,		CONFIG : 'N U T, 0, 0, 0',
	X =  -24.422  mm,	Y =   -338.706  mm,	Z =   -236.046  mm,
	W =  90.000 deg,	P =   0.000 deg,	R =   90.000 deg
};
P[955]{
   GP1:
	UF : 0, UT : 6,		CONFIG : 'N U T, 0, 0, 0',
	X =  -26.247  mm,	Y =   -339.810  mm,	Z =   -236.165  mm,
	W =  90.000 deg,	P =   0.000 deg,	R =   90.000 deg
};
P[956]{
   GP1:
	UF : 0, UT : 6,		CONFIG : 'N U T, 0, 0, 0',
	X =  -27.699  mm,	Y =   -340.524  mm,	Z =   -235.863  mm,
	W =  90.000 deg,	P =   0.000 deg,	R =   90.000 deg
};
P[957]{
   GP1:
	UF : 0, UT : 6,		CONFIG : 'N U T, 0, 0, 0',
	X =  -28.443  mm,	Y =   -341.096  mm,	Z =   -236.208  mm,
	W =  90.000 deg,	P =   0.000 deg,	R =   90.000 deg
};
P[958]{
   GP1:
	UF : 0, UT : 6,		CONFIG : 'N U T, 0, 0, 0',
	X =  -29.759  mm,	Y =   -341.783  mm,	Z =   -236.033  mm,
	W =  90.000 deg,	P =   0.000 deg,	R =   90.000 deg
};
P[959]{
   GP1:
	UF : 0, UT : 6,		CONFIG : 'N U T, 0, 0, 0',
	X =  -33.872  mm,	Y =   -344.199  mm,	Z =   -236.132  mm,
	W =  90.000 deg,	P =   0.000 deg,	R =   90.000 deg
};
P[960]{
   GP1:
	UF : 0, UT : 6,		CONFIG : 'N U T, 0, 0, 0',
	X =  -35.179  mm,	Y =   -344.979  mm,	Z =   -236.195  mm,
	W =  90.000 deg,	P =   0.000 deg,	R =   90.000 deg
};
P[961]{
   GP1:
	UF : 0, UT : 6,		CONFIG : 'N U T, 0, 0, 0',
	X =  -36.184  mm,	Y =   -345.583  mm,	Z =   -236.250  mm,
	W =  90.000 deg,	P =   0.000 deg,	R =   90.000 deg
};
P[962]{
   GP1:
	UF : 0, UT : 6,		CONFIG : 'N U T, 0, 0, 0',
	X =  -37.144  mm,	Y =   -346.035  mm,	Z =   -236.003  mm,
	W =  90.000 deg,	P =   0.000 deg,	R =   90.000 deg
};
P[963]{
   GP1:
	UF : 0, UT : 6,		CONFIG : 'N U T, 0, 0, 0',
	X =  -41.185  mm,	Y =   -348.386  mm,	Z =   -236.046  mm,
	W =  90.000 deg,	P =   0.000 deg,	R =   90.000 deg
};
P[964]{
   GP1:
	UF : 0, UT : 6,		CONFIG : 'N U T, 0, 0, 0',
	X =  -43.367  mm,	Y =   -349.704  mm,	Z =   -236.185  mm,
	W =  90.000 deg,	P =   0.000 deg,	R =   90.000 deg
};
P[965]{
   GP1:
	UF : 0, UT : 6,		CONFIG : 'N U T, 0, 0, 0',
	X =  -46.614  mm,	Y =   -351.503  mm,	Z =   -236.004  mm,
	W =  90.000 deg,	P =   0.000 deg,	R =   90.000 deg
};
P[966]{
   GP1:
	UF : 0, UT : 6,		CONFIG : 'N U T, 0, 0, 0',
	X =  -47.576  mm,	Y =   -352.098  mm,	Z =   -236.099  mm,
	W =  90.000 deg,	P =   0.000 deg,	R =   90.000 deg
};
P[967]{
   GP1:
	UF : 0, UT : 6,		CONFIG : 'N U T, 0, 0, 0',
	X =  -48.390  mm,	Y =   -352.636  mm,	Z =   -236.264  mm,
	W =  90.000 deg,	P =   0.000 deg,	R =   90.000 deg
};
P[968]{
   GP1:
	UF : 0, UT : 6,		CONFIG : 'N U T, 0, 0, 0',
	X =  -49.699  mm,	Y =   -353.301  mm,	Z =   -236.045  mm,
	W =  90.000 deg,	P =   0.000 deg,	R =   90.000 deg
};
P[969]{
   GP1:
	UF : 0, UT : 6,		CONFIG : 'N U T, 0, 0, 0',
	X =  -53.773  mm,	Y =   -355.585  mm,	Z =   -235.877  mm,
	W =  90.000 deg,	P =   0.000 deg,	R =   90.000 deg
};
P[970]{
   GP1:
	UF : 0, UT : 6,		CONFIG : 'N U T, 0, 0, 0',
	X =  -55.873  mm,	Y =   -356.874  mm,	Z =   -236.063  mm,
	W =  90.000 deg,	P =   0.000 deg,	R =   90.000 deg
};
P[971]{
   GP1:
	UF : 0, UT : 6,		CONFIG : 'N U T, 0, 0, 0',
	X =  -57.389  mm,	Y =   -357.741  mm,	Z =   -236.045  mm,
	W =  90.000 deg,	P =   0.000 deg,	R =   90.000 deg
};
P[972]{
   GP1:
	UF : 0, UT : 6,		CONFIG : 'N U T, 0, 0, 0',
	X =  -58.368  mm,	Y =   -358.206  mm,	Z =   -235.800  mm,
	W =  90.000 deg,	P =   0.000 deg,	R =   90.000 deg
};
P[973]{
   GP1:
	UF : 0, UT : 6,		CONFIG : 'N U T, 0, 0, 0',
	X =  -58.889  mm,	Y =   -358.594  mm,	Z =   -236.012  mm,
	W =  90.000 deg,	P =   0.000 deg,	R =   90.000 deg
};
P[974]{
   GP1:
	UF : 0, UT : 6,		CONFIG : 'N U T, 0, 0, 0',
	X =  -60.887  mm,	Y =   -359.742  mm,	Z =   -236.000  mm,
	W =  90.000 deg,	P =   0.000 deg,	R =   90.000 deg
};
P[975]{
   GP1:
	UF : 0, UT : 6,		CONFIG : 'N U T, 0, 0, 0',
	X =  -61.756  mm,	Y =   -360.269  mm,	Z =   -236.061  mm,
	W =  90.000 deg,	P =   0.000 deg,	R =   90.000 deg
};
P[976]{
   GP1:
	UF : 0, UT : 6,		CONFIG : 'N U T, 0, 0, 0',
	X =  -63.843  mm,	Y =   -361.545  mm,	Z =   -236.231  mm,
	W =  90.000 deg,	P =   0.000 deg,	R =   90.000 deg
};
P[977]{
   GP1:
	UF : 0, UT : 6,		CONFIG : 'N U T, 0, 0, 0',
	X =  -64.633  mm,	Y =   -362.004  mm,	Z =   -236.238  mm,
	W =  90.000 deg,	P =   0.000 deg,	R =   90.000 deg
};
P[978]{
   GP1:
	UF : 0, UT : 6,		CONFIG : 'N U T, 0, 0, 0',
	X =  -66.059  mm,	Y =   -362.766  mm,	Z =   -236.090  mm,
	W =  90.000 deg,	P =   0.000 deg,	R =   90.000 deg
};
P[979]{
   GP1:
	UF : 0, UT : 6,		CONFIG : 'N U T, 0, 0, 0',
	X =  -67.088  mm,	Y =   -363.385  mm,	Z =   -236.150  mm,
	W =  90.000 deg,	P =   0.000 deg,	R =   90.000 deg
};
P[980]{
   GP1:
	UF : 0, UT : 6,		CONFIG : 'N U T, 0, 0, 0',
	X =  -69.593  mm,	Y =   -364.812  mm,	Z =   -236.101  mm,
	W =  90.000 deg,	P =   0.000 deg,	R =   90.000 deg
};
P[981]{
   GP1:
	UF : 0, UT : 6,		CONFIG : 'N U T, 0, 0, 0',
	X =  -70.266  mm,	Y =   -365.266  mm,	Z =   -236.262  mm,
	W =  90.000 deg,	P =   0.000 deg,	R =   90.000 deg
};
P[982]{
   GP1:
	UF : 0, UT : 6,		CONFIG : 'N U T, 0, 0, 0',
	X =  -71.199  mm,	Y =   -365.644  mm,	Z =   -235.873  mm,
	W =  90.000 deg,	P =   0.000 deg,	R =   90.000 deg
};
P[983]{
   GP1:
	UF : 0, UT : 6,		CONFIG : 'N U T, 0, 0, 0',
	X =  -72.084  mm,	Y =   -366.311  mm,	Z =   -236.250  mm,
	W =  90.000 deg,	P =   0.000 deg,	R =   90.000 deg
};
P[984]{
   GP1:
	UF : 0, UT : 6,		CONFIG : 'N U T, 0, 0, 0',
	X =  -74.079  mm,	Y =   -367.430  mm,	Z =   -236.171  mm,
	W =  90.000 deg,	P =   0.000 deg,	R =   90.000 deg
};
P[985]{
   GP1:
	UF : 0, UT : 6,		CONFIG : 'N U T, 0, 0, 0',
	X =  -76.920  mm,	Y =   -369.101  mm,	Z =   -236.246  mm,
	W =  90.000 deg,	P =   0.000 deg,	R =   90.000 deg
};
P[986]{
   GP1:
	UF : 0, UT : 6,		CONFIG : 'N U T, 0, 0, 0',
	X =  -77.565  mm,	Y =   -369.370  mm,	Z =   -235.993  mm,
	W =  90.000 deg,	P =   0.000 deg,	R =   90.000 deg
};
P[987]{
   GP1:
	UF : 0, UT : 6,		CONFIG : 'N U T, 0, 0, 0',
	X =  -80.758  mm,	Y =   -371.230  mm,	Z =   -236.035  mm,
	W =  90.000 deg,	P =   0.000 deg,	R =   90.000 deg
};
P[988]{
   GP1:
	UF : 0, UT : 6,		CONFIG : 'N U T, 0, 0, 0',
	X =  -81.525  mm,	Y =   -371.759  mm,	Z =   -236.243  mm,
	W =  90.000 deg,	P =   0.000 deg,	R =   90.000 deg
};
P[989]{
   GP1:
	UF : 0, UT : 6,		CONFIG : 'N U T, 0, 0, 0',
	X =  -83.678  mm,	Y =   -372.932  mm,	Z =   -236.073  mm,
	W =  90.000 deg,	P =   0.000 deg,	R =   90.000 deg
};
P[990]{
   GP1:
	UF : 0, UT : 6,		CONFIG : 'N U T, 0, 0, 0',
	X =  -84.931  mm,	Y =   -373.643  mm,	Z =   -236.041  mm,
	W =  90.000 deg,	P =   0.000 deg,	R =   90.000 deg
};
P[991]{
   GP1:
	UF : 0, UT : 6,		CONFIG : 'N U T, 0, 0, 0',
	X =  -88.701  mm,	Y =   -375.855  mm,	Z =   -236.127  mm,
	W =  90.000 deg,	P =   0.000 deg,	R =   90.000 deg
};
P[992]{
   GP1:
	UF : 0, UT : 6,		CONFIG : 'N U T, 0, 0, 0',
	X =  -89.520  mm,	Y =   -376.336  mm,	Z =   -236.147  mm,
	W =  90.000 deg,	P =   0.000 deg,	R =   90.000 deg
};
P[993]{
   GP1:
	UF : 0, UT : 6,		CONFIG : 'N U T, 0, 0, 0',
	X =  -92.013  mm,	Y =   -377.643  mm,	Z =   -235.826  mm,
	W =  90.000 deg,	P =   0.000 deg,	R =   90.000 deg
};
P[994]{
   GP1:
	UF : 0, UT : 6,		CONFIG : 'N U T, 0, 0, 0',
	X =  -92.458  mm,	Y =   -378.073  mm,	Z =   -236.243  mm,
	W =  90.000 deg,	P =   0.000 deg,	R =   90.000 deg
};
P[995]{
   GP1:
	UF : 0, UT : 6,		CONFIG : 'N U T, 0, 0, 0',
	X =  -95.718  mm,	Y =   -379.898  mm,	Z =   -236.108  mm,
	W =  90.000 deg,	P =   0.000 deg,	R =   90.000 deg
};
P[996]{
   GP1:
	UF : 0, UT : 6,		CONFIG : 'N U T, 0, 0, 0',
	X =  -98.445  mm,	Y =   -381.377  mm,	Z =   -235.876  mm,
	W =  90.000 deg,	P =   0.000 deg,	R =   90.000 deg
};
P[997]{
   GP1:
	UF : 0, UT : 6,		CONFIG : 'N U T, 0, 0, 0',
	X =  -100.704  mm,	Y =   -382.757  mm,	Z =   -236.057  mm,
	W =  90.000 deg,	P =   0.000 deg,	R =   90.000 deg
};
P[998]{
   GP1:
	UF : 0, UT : 6,		CONFIG : 'N U T, 0, 0, 0',
	X =  -103.078  mm,	Y =   -384.132  mm,	Z =   -236.069  mm,
	W =  90.000 deg,	P =   0.000 deg,	R =   90.000 deg
};
P[999]{
   GP1:
	UF : 0, UT : 6,		CONFIG : 'N U T, 0, 0, 0',
	X =  -103.626  mm,	Y =   -384.519  mm,	Z =   -236.239  mm,
	W =  90.000 deg,	P =   0.000 deg,	R =   90.000 deg
};
P[1000]{
   GP1:
	UF : 0, UT : 6,		CONFIG : 'N U T, 0, 0, 0',
	X =  -104.170  mm,	Y =   -384.655  mm,	Z =   -235.809  mm,
	W =  90.000 deg,	P =   0.000 deg,	R =   90.000 deg
};
P[1001]{
   GP1:
	UF : 0, UT : 6,		CONFIG : 'N U T, 0, 0, 0',
	X =  -105.045  mm,	Y =   -385.205  mm,	Z =   -235.916  mm,
	W =  90.000 deg,	P =   0.000 deg,	R =   90.000 deg
};
P[1002]{
   GP1:
	UF : 0, UT : 6,		CONFIG : 'N U T, 0, 0, 0',
	X =  -107.937  mm,	Y =   -387.012  mm,	Z =   -236.050  mm,
	W =  90.000 deg,	P =   0.000 deg,	R =   90.000 deg
};
P[1003]{
   GP1:
	UF : 0, UT : 6,		CONFIG : 'N U T, 0, 0, 0',
	X =  -109.477  mm,	Y =   -388.233  mm,	Z =   -236.264  mm,
	W =  90.000 deg,	P =   0.000 deg,	R =   90.000 deg
};
P[1004]{
   GP1:
	UF : 0, UT : 6,		CONFIG : 'N U T, 0, 0, 0',
	X =  -111.371  mm,	Y =   -390.174  mm,	Z =   -236.067  mm,
	W =  90.000 deg,	P =   0.000 deg,	R =   90.000 deg
};
P[1005]{
   GP1:
	UF : 0, UT : 6,		CONFIG : 'N U T, 0, 0, 0',
	X =  -112.980  mm,	Y =   -392.701  mm,	Z =   -235.796  mm,
	W =  90.000 deg,	P =   0.000 deg,	R =   90.000 deg
};
P[1006]{
   GP1:
	UF : 0, UT : 6,		CONFIG : 'N U T, 0, 0, 0',
	X =  -113.381  mm,	Y =   -394.197  mm,	Z =   -235.989  mm,
	W =  90.000 deg,	P =   0.000 deg,	R =   90.000 deg
};
P[1007]{
   GP1:
	UF : 0, UT : 6,		CONFIG : 'N U T, 0, 0, 0',
	X =  -113.744  mm,	Y =   -396.720  mm,	Z =   -236.164  mm,
	W =  90.000 deg,	P =   0.000 deg,	R =   90.000 deg
};
P[1008]{
   GP1:
	UF : 0, UT : 6,		CONFIG : 'N U T, 0, 0, 0',
	X =  -113.839  mm,	Y =   -397.587  mm,	Z =   -236.024  mm,
	W =  90.000 deg,	P =   0.000 deg,	R =   90.000 deg
};
P[1009]{
   GP1:
	UF : 0, UT : 6,		CONFIG : 'N U T, 0, 0, 0',
	X =  -113.840  mm,	Y =   -398.707  mm,	Z =   -235.966  mm,
	W =  90.000 deg,	P =   0.000 deg,	R =   90.000 deg
};
P[1010]{
   GP1:
	UF : 0, UT : 6,		CONFIG : 'N U T, 0, 0, 0',
	X =  -113.375  mm,	Y =   -400.617  mm,	Z =   -236.228  mm,
	W =  90.000 deg,	P =   0.000 deg,	R =   90.000 deg
};
P[1011]{
   GP1:
	UF : 0, UT : 6,		CONFIG : 'N U T, 0, 0, 0',
	X =  -113.238  mm,	Y =   -401.276  mm,	Z =   -236.175  mm,
	W =  90.000 deg,	P =   0.000 deg,	R =   90.000 deg
};
P[1012]{
   GP1:
	UF : 0, UT : 6,		CONFIG : 'N U T, 0, 0, 0',
	X =  -112.672  mm,	Y =   -402.709  mm,	Z =   -236.203  mm,
	W =  90.000 deg,	P =   0.000 deg,	R =   90.000 deg
};
P[1013]{
   GP1:
	UF : 0, UT : 6,		CONFIG : 'N U T, 0, 0, 0',
	X =  -112.409  mm,	Y =   -403.378  mm,	Z =   -236.119  mm,
	W =  90.000 deg,	P =   0.000 deg,	R =   90.000 deg
};
P[1014]{
   GP1:
	UF : 0, UT : 6,		CONFIG : 'N U T, 0, 0, 0',
	X =  -112.161  mm,	Y =   -403.997  mm,	Z =   -236.030  mm,
	W =  90.000 deg,	P =   0.000 deg,	R =   90.000 deg
};
P[1015]{
   GP1:
	UF : 0, UT : 6,		CONFIG : 'N U T, 0, 0, 0',
	X =  -111.868  mm,	Y =   -404.599  mm,	Z =   -235.968  mm,
	W =  90.000 deg,	P =   0.000 deg,	R =   90.000 deg
};
P[1016]{
   GP1:
	UF : 0, UT : 6,		CONFIG : 'N U T, 0, 0, 0',
	X =  -110.358  mm,	Y =   -407.079  mm,	Z =   -236.155  mm,
	W =  90.000 deg,	P =   0.000 deg,	R =   90.000 deg
};
P[1017]{
   GP1:
	UF : 0, UT : 6,		CONFIG : 'N U T, 0, 0, 0',
	X =  -109.510  mm,	Y =   -408.483  mm,	Z =   -236.247  mm,
	W =  90.000 deg,	P =   0.000 deg,	R =   90.000 deg
};
P[1018]{
   GP1:
	UF : 0, UT : 6,		CONFIG : 'N U T, 0, 0, 0',
	X =  -108.918  mm,	Y =   -409.550  mm,	Z =   -236.188  mm,
	W =  90.000 deg,	P =   0.000 deg,	R =   90.000 deg
};
P[1019]{
   GP1:
	UF : 0, UT : 6,		CONFIG : 'N U T, 0, 0, 0',
	X =  -107.155  mm,	Y =   -412.900  mm,	Z =   -235.773  mm,
	W =  90.000 deg,	P =   0.000 deg,	R =   90.000 deg
};
P[1020]{
   GP1:
	UF : 0, UT : 6,		CONFIG : 'N U T, 0, 0, 0',
	X =  -106.210  mm,	Y =   -414.224  mm,	Z =   -236.210  mm,
	W =  90.000 deg,	P =   0.000 deg,	R =   90.000 deg
};
P[1021]{
   GP1:
	UF : 0, UT : 6,		CONFIG : 'N U T, 0, 0, 0',
	X =  -104.525  mm,	Y =   -417.380  mm,	Z =   -235.877  mm,
	W =  90.000 deg,	P =   0.000 deg,	R =   90.000 deg
};
P[1022]{
   GP1:
	UF : 0, UT : 6,		CONFIG : 'N U T, 0, 0, 0',
	X =  -103.037  mm,	Y =   -419.751  mm,	Z =   -236.166  mm,
	W =  90.000 deg,	P =   0.000 deg,	R =   90.000 deg
};
P[1023]{
   GP1:
	UF : 0, UT : 6,		CONFIG : 'N U T, 0, 0, 0',
	X =  -102.463  mm,	Y =   -420.740  mm,	Z =   -236.173  mm,
	W =  90.000 deg,	P =   0.000 deg,	R =   90.000 deg
};
P[1024]{
   GP1:
	UF : 0, UT : 6,		CONFIG : 'N U T, 0, 0, 0',
	X =  -101.858  mm,	Y =   -421.750  mm,	Z =   -236.227  mm,
	W =  90.000 deg,	P =   0.000 deg,	R =   90.000 deg
};
P[1025]{
   GP1:
	UF : 0, UT : 6,		CONFIG : 'N U T, 0, 0, 0',
	X =  -100.640  mm,	Y =   -423.858  mm,	Z =   -236.231  mm,
	W =  90.000 deg,	P =   0.000 deg,	R =   90.000 deg
};
P[1026]{
   GP1:
	UF : 0, UT : 6,		CONFIG : 'N U T, 0, 0, 0',
	X =  -100.236  mm,	Y =   -424.631  mm,	Z =   -236.125  mm,
	W =  90.000 deg,	P =   0.000 deg,	R =   90.000 deg
};
P[1027]{
   GP1:
	UF : 0, UT : 6,		CONFIG : 'N U T, 0, 0, 0',
	X =  -99.855  mm,	Y =   -425.220  mm,	Z =   -236.223  mm,
	W =  90.000 deg,	P =   0.000 deg,	R =   90.000 deg
};
P[1028]{
   GP1:
	UF : 0, UT : 6,		CONFIG : 'N U T, 0, 0, 0',
	X =  -98.709  mm,	Y =   -427.305  mm,	Z =   -236.085  mm,
	W =  90.000 deg,	P =   0.000 deg,	R =   90.000 deg
};
P[1029]{
   GP1:
	UF : 0, UT : 6,		CONFIG : 'N U T, 0, 0, 0',
	X =  -98.058  mm,	Y =   -428.506  mm,	Z =   -235.982  mm,
	W =  90.000 deg,	P =   0.000 deg,	R =   90.000 deg
};
P[1030]{
   GP1:
	UF : 0, UT : 6,		CONFIG : 'N U T, 0, 0, 0',
	X =  -97.307  mm,	Y =   -429.925  mm,	Z =   -235.818  mm,
	W =  90.000 deg,	P =   0.000 deg,	R =   90.000 deg
};
P[1031]{
   GP1:
	UF : 0, UT : 6,		CONFIG : 'N U T, 0, 0, 0',
	X =  -96.671  mm,	Y =   -430.737  mm,	Z =   -236.222  mm,
	W =  90.000 deg,	P =   0.000 deg,	R =   90.000 deg
};
P[1032]{
   GP1:
	UF : 0, UT : 6,		CONFIG : 'N U T, 0, 0, 0',
	X =  -96.043  mm,	Y =   -431.823  mm,	Z =   -236.224  mm,
	W =  90.000 deg,	P =   0.000 deg,	R =   90.000 deg
};
P[1033]{
   GP1:
	UF : 0, UT : 6,		CONFIG : 'N U T, 0, 0, 0',
	X =  -95.155  mm,	Y =   -433.333  mm,	Z =   -236.263  mm,
	W =  90.000 deg,	P =   0.000 deg,	R =   90.000 deg
};
P[1034]{
   GP1:
	UF : 0, UT : 6,		CONFIG : 'N U T, 0, 0, 0',
	X =  -94.895  mm,	Y =   -433.981  mm,	Z =   -235.984  mm,
	W =  90.000 deg,	P =   0.000 deg,	R =   90.000 deg
};
P[1035]{
   GP1:
	UF : 0, UT : 6,		CONFIG : 'N U T, 0, 0, 0',
	X =  -94.528  mm,	Y =   -434.604  mm,	Z =   -236.004  mm,
	W =  90.000 deg,	P =   0.000 deg,	R =   90.000 deg
};
P[1036]{
   GP1:
	UF : 0, UT : 6,		CONFIG : 'N U T, 0, 0, 0',
	X =  -93.889  mm,	Y =   -435.573  mm,	Z =   -236.197  mm,
	W =  90.000 deg,	P =   0.000 deg,	R =   90.000 deg
};
P[1037]{
   GP1:
	UF : 0, UT : 6,		CONFIG : 'N U T, 0, 0, 0',
	X =  -92.168  mm,	Y =   -438.666  mm,	Z =   -236.039  mm,
	W =  90.000 deg,	P =   0.000 deg,	R =   90.000 deg
};
P[1038]{
   GP1:
	UF : 0, UT : 6,		CONFIG : 'N U T, 0, 0, 0',
	X =  -91.710  mm,	Y =   -439.309  mm,	Z =   -236.250  mm,
	W =  90.000 deg,	P =   0.000 deg,	R =   90.000 deg
};
P[1039]{
   GP1:
	UF : 0, UT : 6,		CONFIG : 'N U T, 0, 0, 0',
	X =  -90.857  mm,	Y =   -441.122  mm,	Z =   -235.777  mm,
	W =  90.000 deg,	P =   0.000 deg,	R =   90.000 deg
};
P[1040]{
   GP1:
	UF : 0, UT : 6,		CONFIG : 'N U T, 0, 0, 0',
	X =  -89.996  mm,	Y =   -442.490  mm,	Z =   -235.953  mm,
	W =  90.000 deg,	P =   0.000 deg,	R =   90.000 deg
};
P[1041]{
   GP1:
	UF : 0, UT : 6,		CONFIG : 'N U T, 0, 0, 0',
	X =  -89.179  mm,	Y =   -443.708  mm,	Z =   -236.228  mm,
	W =  90.000 deg,	P =   0.000 deg,	R =   90.000 deg
};
P[1042]{
   GP1:
	UF : 0, UT : 6,		CONFIG : 'N U T, 0, 0, 0',
	X =  -88.804  mm,	Y =   -444.592  mm,	Z =   -235.897  mm,
	W =  90.000 deg,	P =   0.000 deg,	R =   90.000 deg
};
P[1043]{
   GP1:
	UF : 0, UT : 6,		CONFIG : 'N U T, 0, 0, 0',
	X =  -87.422  mm,	Y =   -446.789  mm,	Z =   -236.176  mm,
	W =  90.000 deg,	P =   0.000 deg,	R =   90.000 deg
};
P[1044]{
   GP1:
	UF : 0, UT : 6,		CONFIG : 'N U T, 0, 0, 0',
	X =  -86.971  mm,	Y =   -447.570  mm,	Z =   -236.175  mm,
	W =  90.000 deg,	P =   0.000 deg,	R =   90.000 deg
};
P[1045]{
   GP1:
	UF : 0, UT : 6,		CONFIG : 'N U T, 0, 0, 0',
	X =  -86.175  mm,	Y =   -449.096  mm,	Z =   -235.968  mm,
	W =  90.000 deg,	P =   0.000 deg,	R =   90.000 deg
};
P[1046]{
   GP1:
	UF : 0, UT : 6,		CONFIG : 'N U T, 0, 0, 0',
	X =  -85.177  mm,	Y =   -450.759  mm,	Z =   -236.059  mm,
	W =  90.000 deg,	P =   0.000 deg,	R =   90.000 deg
};
P[1047]{
   GP1:
	UF : 0, UT : 6,		CONFIG : 'N U T, 0, 0, 0',
	X =  -83.376  mm,	Y =   -453.914  mm,	Z =   -236.009  mm,
	W =  90.000 deg,	P =   0.000 deg,	R =   90.000 deg
};
P[1048]{
   GP1:
	UF : 0, UT : 6,		CONFIG : 'N U T, 0, 0, 0',
	X =  -82.039  mm,	Y =   -456.079  mm,	Z =   -236.222  mm,
	W =  90.000 deg,	P =   0.000 deg,	R =   90.000 deg
};
P[1049]{
   GP1:
	UF : 0, UT : 6,		CONFIG : 'N U T, 0, 0, 0',
	X =  -81.484  mm,	Y =   -457.083  mm,	Z =   -236.160  mm,
	W =  90.000 deg,	P =   0.000 deg,	R =   90.000 deg
};
P[1050]{
   GP1:
	UF : 0, UT : 6,		CONFIG : 'N U T, 0, 0, 0',
	X =  -80.295  mm,	Y =   -459.325  mm,	Z =   -235.905  mm,
	W =  90.000 deg,	P =   0.000 deg,	R =   90.000 deg
};
P[1051]{
   GP1:
	UF : 0, UT : 6,		CONFIG : 'N U T, 0, 0, 0',
	X =  -77.772  mm,	Y =   -463.443  mm,	Z =   -236.257  mm,
	W =  90.000 deg,	P =   0.000 deg,	R =   90.000 deg
};
P[1052]{
   GP1:
	UF : 0, UT : 6,		CONFIG : 'N U T, 0, 0, 0',
	X =  -77.411  mm,	Y =   -464.162  mm,	Z =   -236.125  mm,
	W =  90.000 deg,	P =   0.000 deg,	R =   90.000 deg
};
P[1053]{
   GP1:
	UF : 0, UT : 6,		CONFIG : 'N U T, 0, 0, 0',
	X =  -76.719  mm,	Y =   -465.602  mm,	Z =   -235.789  mm,
	W =  90.000 deg,	P =   0.000 deg,	R =   90.000 deg
};
P[1054]{
   GP1:
	UF : 0, UT : 6,		CONFIG : 'N U T, 0, 0, 0',
	X =  -75.722  mm,	Y =   -467.174  mm,	Z =   -236.004  mm,
	W =  90.000 deg,	P =   0.000 deg,	R =   90.000 deg
};
P[1055]{
   GP1:
	UF : 0, UT : 6,		CONFIG : 'N U T, 0, 0, 0',
	X =  -75.102  mm,	Y =   -468.210  mm,	Z =   -236.057  mm,
	W =  90.000 deg,	P =   0.000 deg,	R =   90.000 deg
};
P[1056]{
   GP1:
	UF : 0, UT : 6,		CONFIG : 'N U T, 0, 0, 0',
	X =  -74.529  mm,	Y =   -469.095  mm,	Z =   -236.209  mm,
	W =  90.000 deg,	P =   0.000 deg,	R =   90.000 deg
};
P[1057]{
   GP1:
	UF : 0, UT : 6,		CONFIG : 'N U T, 0, 0, 0',
	X =  -73.752  mm,	Y =   -470.472  mm,	Z =   -236.164  mm,
	W =  90.000 deg,	P =   0.000 deg,	R =   90.000 deg
};
P[1058]{
   GP1:
	UF : 0, UT : 6,		CONFIG : 'N U T, 0, 0, 0',
	X =  -72.781  mm,	Y =   -472.257  mm,	Z =   -236.022  mm,
	W =  90.000 deg,	P =   0.000 deg,	R =   90.000 deg
};
P[1059]{
   GP1:
	UF : 0, UT : 6,		CONFIG : 'N U T, 0, 0, 0',
	X =  -72.262  mm,	Y =   -473.021  mm,	Z =   -236.209  mm,
	W =  90.000 deg,	P =   0.000 deg,	R =   90.000 deg
};
P[1060]{
   GP1:
	UF : 0, UT : 6,		CONFIG : 'N U T, 0, 0, 0',
	X =  -71.019  mm,	Y =   -475.346  mm,	Z =   -235.969  mm,
	W =  90.000 deg,	P =   0.000 deg,	R =   90.000 deg
};
P[1061]{
   GP1:
	UF : 0, UT : 6,		CONFIG : 'N U T, 0, 0, 0',
	X =  -70.675  mm,	Y =   -475.901  mm,	Z =   -236.025  mm,
	W =  90.000 deg,	P =   0.000 deg,	R =   90.000 deg
};
P[1062]{
   GP1:
	UF : 0, UT : 6,		CONFIG : 'N U T, 0, 0, 0',
	X =  -70.094  mm,	Y =   -476.837  mm,	Z =   -236.122  mm,
	W =  90.000 deg,	P =   0.000 deg,	R =   90.000 deg
};
P[1063]{
   GP1:
	UF : 0, UT : 6,		CONFIG : 'N U T, 0, 0, 0',
	X =  -69.054  mm,	Y =   -478.562  mm,	Z =   -236.229  mm,
	W =  90.000 deg,	P =   0.000 deg,	R =   90.000 deg
};
P[1064]{
   GP1:
	UF : 0, UT : 6,		CONFIG : 'N U T, 0, 0, 0',
	X =  -68.650  mm,	Y =   -479.532  mm,	Z =   -235.849  mm,
	W =  90.000 deg,	P =   0.000 deg,	R =   90.000 deg
};
P[1065]{
   GP1:
	UF : 0, UT : 6,		CONFIG : 'N U T, 0, 0, 0',
	X =  -67.807  mm,	Y =   -480.822  mm,	Z =   -236.089  mm,
	W =  90.000 deg,	P =   0.000 deg,	R =   90.000 deg
};
P[1066]{
   GP1:
	UF : 0, UT : 6,		CONFIG : 'N U T, 0, 0, 0',
	X =  -67.431  mm,	Y =   -481.514  mm,	Z =   -236.032  mm,
	W =  90.000 deg,	P =   0.000 deg,	R =   90.000 deg
};
P[1067]{
   GP1:
	UF : 0, UT : 6,		CONFIG : 'N U T, 0, 0, 0',
	X =  -65.275  mm,	Y =   -485.125  mm,	Z =   -236.203  mm,
	W =  90.000 deg,	P =   0.000 deg,	R =   90.000 deg
};
P[1068]{
   GP1:
	UF : 0, UT : 6,		CONFIG : 'N U T, 0, 0, 0',
	X =  -64.367  mm,	Y =   -486.700  mm,	Z =   -236.201  mm,
	W =  90.000 deg,	P =   0.000 deg,	R =   90.000 deg
};
P[1069]{
   GP1:
	UF : 0, UT : 6,		CONFIG : 'N U T, 0, 0, 0',
	X =  -63.658  mm,	Y =   -488.093  mm,	Z =   -235.970  mm,
	W =  90.000 deg,	P =   0.000 deg,	R =   90.000 deg
};
P[1070]{
   GP1:
	UF : 0, UT : 6,		CONFIG : 'N U T, 0, 0, 0',
	X =  -62.922  mm,	Y =   -489.176  mm,	Z =   -236.240  mm,
	W =  90.000 deg,	P =   0.000 deg,	R =   90.000 deg
};
P[1071]{
   GP1:
	UF : 0, UT : 6,		CONFIG : 'N U T, 0, 0, 0',
	X =  -62.236  mm,	Y =   -490.359  mm,	Z =   -236.247  mm,
	W =  90.000 deg,	P =   0.000 deg,	R =   90.000 deg
};
P[1072]{
   GP1:
	UF : 0, UT : 6,		CONFIG : 'N U T, 0, 0, 0',
	X =  -61.709  mm,	Y =   -491.421  mm,	Z =   -236.038  mm,
	W =  90.000 deg,	P =   0.000 deg,	R =   90.000 deg
};
P[1073]{
   GP1:
	UF : 0, UT : 6,		CONFIG : 'N U T, 0, 0, 0',
	X =  -61.214  mm,	Y =   -492.216  mm,	Z =   -236.125  mm,
	W =  90.000 deg,	P =   0.000 deg,	R =   90.000 deg
};
P[1074]{
   GP1:
	UF : 0, UT : 6,		CONFIG : 'N U T, 0, 0, 0',
	X =  -60.818  mm,	Y =   -493.043  mm,	Z =   -235.927  mm,
	W =  90.000 deg,	P =   0.000 deg,	R =   90.000 deg
};
P[1075]{
   GP1:
	UF : 0, UT : 6,		CONFIG : 'N U T, 0, 0, 0',
	X =  -59.507  mm,	Y =   -495.107  mm,	Z =   -236.217  mm,
	W =  90.000 deg,	P =   0.000 deg,	R =   90.000 deg
};
P[1076]{
   GP1:
	UF : 0, UT : 6,		CONFIG : 'N U T, 0, 0, 0',
	X =  -58.939  mm,	Y =   -496.136  mm,	Z =   -236.152  mm,
	W =  90.000 deg,	P =   0.000 deg,	R =   90.000 deg
};
P[1077]{
   GP1:
	UF : 0, UT : 6,		CONFIG : 'N U T, 0, 0, 0',
	X =  -56.466  mm,	Y =   -500.548  mm,	Z =   -235.971  mm,
	W =  90.000 deg,	P =   0.000 deg,	R =   90.000 deg
};
P[1078]{
   GP1:
	UF : 0, UT : 6,		CONFIG : 'N U T, 0, 0, 0',
	X =  -56.038  mm,	Y =   -501.284  mm,	Z =   -235.979  mm,
	W =  90.000 deg,	P =   0.000 deg,	R =   90.000 deg
};
P[1079]{
   GP1:
	UF : 0, UT : 6,		CONFIG : 'N U T, 0, 0, 0',
	X =  -55.443  mm,	Y =   -502.184  mm,	Z =   -236.160  mm,
	W =  90.000 deg,	P =   0.000 deg,	R =   90.000 deg
};
P[1080]{
   GP1:
	UF : 0, UT : 6,		CONFIG : 'N U T, 0, 0, 0',
	X =  -54.078  mm,	Y =   -504.696  mm,	Z =   -235.954  mm,
	W =  90.000 deg,	P =   0.000 deg,	R =   90.000 deg
};
P[1081]{
   GP1:
	UF : 0, UT : 6,		CONFIG : 'N U T, 0, 0, 0',
	X =  -52.301  mm,	Y =   -507.713  mm,	Z =   -236.039  mm,
	W =  90.000 deg,	P =   0.000 deg,	R =   90.000 deg
};
P[1082]{
   GP1:
	UF : 0, UT : 6,		CONFIG : 'N U T, 0, 0, 0',
	X =  -49.640  mm,	Y =   -512.446  mm,	Z =   -235.865  mm,
	W =  90.000 deg,	P =   0.000 deg,	R =   90.000 deg
};
P[1083]{
   GP1:
	UF : 0, UT : 6,		CONFIG : 'N U T, 0, 0, 0',
	X =  -48.400  mm,	Y =   -514.635  mm,	Z =   -235.807  mm,
	W =  90.000 deg,	P =   0.000 deg,	R =   90.000 deg
};
P[1084]{
   GP1:
	UF : 0, UT : 6,		CONFIG : 'N U T, 0, 0, 0',
	X =  -48.001  mm,	Y =   -515.132  mm,	Z =   -236.079  mm,
	W =  90.000 deg,	P =   0.000 deg,	R =   90.000 deg
};
P[1085]{
   GP1:
	UF : 0, UT : 6,		CONFIG : 'N U T, 0, 0, 0',
	X =  -46.704  mm,	Y =   -517.366  mm,	Z =   -236.097  mm,
	W =  90.000 deg,	P =   0.000 deg,	R =   90.000 deg
};
P[1086]{
   GP1:
	UF : 0, UT : 6,		CONFIG : 'N U T, 0, 0, 0',
	X =  -46.064  mm,	Y =   -518.460  mm,	Z =   -236.116  mm,
	W =  90.000 deg,	P =   0.000 deg,	R =   90.000 deg
};
P[1087]{
   GP1:
	UF : 0, UT : 6,		CONFIG : 'N U T, 0, 0, 0',
	X =  -45.271  mm,	Y =   -519.771  mm,	Z =   -236.202  mm,
	W =  90.000 deg,	P =   0.000 deg,	R =   90.000 deg
};
P[1088]{
   GP1:
	UF : 0, UT : 6,		CONFIG : 'N U T, 0, 0, 0',
	X =  -42.414  mm,	Y =   -524.955  mm,	Z =   -235.872  mm,
	W =  90.000 deg,	P =   0.000 deg,	R =   90.000 deg
};
P[1089]{
   GP1:
	UF : 0, UT : 6,		CONFIG : 'N U T, 0, 0, 0',
	X =  -40.276  mm,	Y =   -528.381  mm,	Z =   -236.263  mm,
	W =  90.000 deg,	P =   0.000 deg,	R =   90.000 deg
};
P[1090]{
   GP1:
	UF : 0, UT : 6,		CONFIG : 'N U T, 0, 0, 0',
	X =  -39.072  mm,	Y =   -530.482  mm,	Z =   -236.241  mm,
	W =  90.000 deg,	P =   0.000 deg,	R =   90.000 deg
};
P[1091]{
   GP1:
	UF : 0, UT : 6,		CONFIG : 'N U T, 0, 0, 0',
	X =  -35.519  mm,	Y =   -536.717  mm,	Z =   -236.124  mm,
	W =  90.000 deg,	P =   0.000 deg,	R =   90.000 deg
};
P[1092]{
   GP1:
	UF : 0, UT : 6,		CONFIG : 'N U T, 0, 0, 0',
	X =  -34.699  mm,	Y =   -538.267  mm,	Z =   -235.944  mm,
	W =  90.000 deg,	P =   0.000 deg,	R =   90.000 deg
};
P[1093]{
   GP1:
	UF : 0, UT : 6,		CONFIG : 'N U T, 0, 0, 0',
	X =  -34.121  mm,	Y =   -539.290  mm,	Z =   -235.911  mm,
	W =  90.000 deg,	P =   0.000 deg,	R =   90.000 deg
};
P[1094]{
   GP1:
	UF : 0, UT : 6,		CONFIG : 'N U T, 0, 0, 0',
	X =  -32.478  mm,	Y =   -542.011  mm,	Z =   -236.085  mm,
	W =  90.000 deg,	P =   0.000 deg,	R =   90.000 deg
};
P[1095]{
   GP1:
	UF : 0, UT : 6,		CONFIG : 'N U T, 0, 0, 0',
	X =  -31.969  mm,	Y =   -542.984  mm,	Z =   -235.957  mm,
	W =  90.000 deg,	P =   0.000 deg,	R =   90.000 deg
};
P[1096]{
   GP1:
	UF : 0, UT : 6,		CONFIG : 'N U T, 0, 0, 0',
	X =  -30.735  mm,	Y =   -544.923  mm,	Z =   -236.236  mm,
	W =  90.000 deg,	P =   0.000 deg,	R =   90.000 deg
};
P[1097]{
   GP1:
	UF : 0, UT : 6,		CONFIG : 'N U T, 0, 0, 0',
	X =  -29.634  mm,	Y =   -546.926  mm,	Z =   -236.101  mm,
	W =  90.000 deg,	P =   0.000 deg,	R =   90.000 deg
};
P[1098]{
   GP1:
	UF : 0, UT : 6,		CONFIG : 'N U T, 0, 0, 0',
	X =  -29.319  mm,	Y =   -547.675  mm,	Z =   -235.816  mm,
	W =  90.000 deg,	P =   0.000 deg,	R =   90.000 deg
};
P[1099]{
   GP1:
	UF : 0, UT : 6,		CONFIG : 'N U T, 0, 0, 0',
	X =  -28.280  mm,	Y =   -549.251  mm,	Z =   -236.129  mm,
	W =  90.000 deg,	P =   0.000 deg,	R =   90.000 deg
};
P[1100]{
   GP1:
	UF : 0, UT : 6,		CONFIG : 'N U T, 0, 0, 0',
	X =  -27.810  mm,	Y =   -550.023  mm,	Z =   -236.187  mm,
	W =  90.000 deg,	P =   0.000 deg,	R =   90.000 deg
};
P[1101]{
   GP1:
	UF : 0, UT : 6,		CONFIG : 'N U T, 0, 0, 0',
	X =  -27.412  mm,	Y =   -550.878  mm,	Z =   -235.957  mm,
	W =  90.000 deg,	P =   0.000 deg,	R =   90.000 deg
};
P[1102]{
   GP1:
	UF : 0, UT : 6,		CONFIG : 'N U T, 0, 0, 0',
	X =  -26.931  mm,	Y =   -551.535  mm,	Z =   -236.204  mm,
	W =  90.000 deg,	P =   0.000 deg,	R =   90.000 deg
};
P[1103]{
   GP1:
	UF : 0, UT : 6,		CONFIG : 'N U T, 0, 0, 0',
	X =  -25.948  mm,	Y =   -553.204  mm,	Z =   -236.250  mm,
	W =  90.000 deg,	P =   0.000 deg,	R =   90.000 deg
};
P[1104]{
   GP1:
	UF : 0, UT : 6,		CONFIG : 'N U T, 0, 0, 0',
	X =  -25.090  mm,	Y =   -554.958  mm,	Z =   -235.874  mm,
	W =  90.000 deg,	P =   0.000 deg,	R =   90.000 deg
};
P[1105]{
   GP1:
	UF : 0, UT : 6,		CONFIG : 'N U T, 0, 0, 0',
	X =  -21.250  mm,	Y =   -561.344  mm,	Z =   -236.245  mm,
	W =  90.000 deg,	P =   0.000 deg,	R =   90.000 deg
};
P[1106]{
   GP1:
	UF : 0, UT : 6,		CONFIG : 'N U T, 0, 0, 0',
	X =  -21.154  mm,	Y =   -561.829  mm,	Z =   -235.799  mm,
	W =  90.000 deg,	P =   0.000 deg,	R =   90.000 deg
};
P[1107]{
   GP1:
	UF : 0, UT : 6,		CONFIG : 'N U T, 0, 0, 0',
	X =  -20.797  mm,	Y =   -562.342  mm,	Z =   -235.948  mm,
	W =  90.000 deg,	P =   0.000 deg,	R =   90.000 deg
};
P[1108]{
   GP1:
	UF : 0, UT : 6,		CONFIG : 'N U T, 0, 0, 0',
	X =  -19.208  mm,	Y =   -564.871  mm,	Z =   -236.259  mm,
	W =  90.000 deg,	P =   0.000 deg,	R =   90.000 deg
};
P[1109]{
   GP1:
	UF : 0, UT : 6,		CONFIG : 'N U T, 0, 0, 0',
	X =  -18.695  mm,	Y =   -565.820  mm,	Z =   -236.172  mm,
	W =  90.000 deg,	P =   0.000 deg,	R =   90.000 deg
};
P[1110]{
   GP1:
	UF : 0, UT : 6,		CONFIG : 'N U T, 0, 0, 0',
	X =  -18.282  mm,	Y =   -566.562  mm,	Z =   -236.137  mm,
	W =  90.000 deg,	P =   0.000 deg,	R =   90.000 deg
};
P[1111]{
   GP1:
	UF : 0, UT : 6,		CONFIG : 'N U T, 0, 0, 0',
	X =  -17.824  mm,	Y =   -567.527  mm,	Z =   -235.894  mm,
	W =  90.000 deg,	P =   0.000 deg,	R =   90.000 deg
};
P[1112]{
   GP1:
	UF : 0, UT : 6,		CONFIG : 'N U T, 0, 0, 0',
	X =  -16.701  mm,	Y =   -569.353  mm,	Z =   -236.062  mm,
	W =  90.000 deg,	P =   0.000 deg,	R =   90.000 deg
};
P[1113]{
   GP1:
	UF : 0, UT : 6,		CONFIG : 'N U T, 0, 0, 0',
	X =  -15.859  mm,	Y =   -570.916  mm,	Z =   -235.917  mm,
	W =  90.000 deg,	P =   0.000 deg,	R =   90.000 deg
};
P[1114]{
   GP1:
	UF : 0, UT : 6,		CONFIG : 'N U T, 0, 0, 0',
	X =  -14.947  mm,	Y =   -572.494  mm,	Z =   -235.916  mm,
	W =  90.000 deg,	P =   0.000 deg,	R =   90.000 deg
};
P[1115]{
   GP1:
	UF : 0, UT : 6,		CONFIG : 'N U T, 0, 0, 0',
	X =  -14.324  mm,	Y =   -573.422  mm,	Z =   -236.129  mm,
	W =  90.000 deg,	P =   0.000 deg,	R =   90.000 deg
};
P[1116]{
   GP1:
	UF : 0, UT : 6,		CONFIG : 'N U T, 0, 0, 0',
	X =  -13.737  mm,	Y =   -574.563  mm,	Z =   -235.956  mm,
	W =  90.000 deg,	P =   0.000 deg,	R =   90.000 deg
};
P[1117]{
   GP1:
	UF : 0, UT : 6,		CONFIG : 'N U T, 0, 0, 0',
	X =  -12.427  mm,	Y =   -576.773  mm,	Z =   -236.037  mm,
	W =  90.000 deg,	P =   0.000 deg,	R =   90.000 deg
};
P[1118]{
   GP1:
	UF : 0, UT : 6,		CONFIG : 'N U T, 0, 0, 0',
	X =  -11.441  mm,	Y =   -578.545  mm,	Z =   -235.948  mm,
	W =  90.000 deg,	P =   0.000 deg,	R =   90.000 deg
};
P[1119]{
   GP1:
	UF : 0, UT : 6,		CONFIG : 'N U T, 0, 0, 0',
	X =  -10.909  mm,	Y =   -579.363  mm,	Z =   -236.093  mm,
	W =  90.000 deg,	P =   0.000 deg,	R =   90.000 deg
};
P[1120]{
   GP1:
	UF : 0, UT : 6,		CONFIG : 'N U T, 0, 0, 0',
	X =  -6.868  mm,	Y =   -586.367  mm,	Z =   -236.084  mm,
	W =  90.000 deg,	P =   0.000 deg,	R =   90.000 deg
};
P[1121]{
   GP1:
	UF : 0, UT : 6,		CONFIG : 'N U T, 0, 0, 0',
	X =  -6.384  mm,	Y =   -587.157  mm,	Z =   -236.154  mm,
	W =  90.000 deg,	P =   0.000 deg,	R =   90.000 deg
};
P[1122]{
   GP1:
	UF : 0, UT : 6,		CONFIG : 'N U T, 0, 0, 0',
	X =  -6.009  mm,	Y =   -587.762  mm,	Z =   -236.215  mm,
	W =  90.000 deg,	P =   0.000 deg,	R =   90.000 deg
};
P[1123]{
   GP1:
	UF : 0, UT : 6,		CONFIG : 'N U T, 0, 0, 0',
	X =  -5.397  mm,	Y =   -588.915  mm,	Z =   -236.085  mm,
	W =  90.000 deg,	P =   0.000 deg,	R =   90.000 deg
};
P[1124]{
   GP1:
	UF : 0, UT : 6,		CONFIG : 'N U T, 0, 0, 0',
	X =  -4.170  mm,	Y =   -591.063  mm,	Z =   -236.051  mm,
	W =  90.000 deg,	P =   0.000 deg,	R =   90.000 deg
};
P[1125]{
   GP1:
	UF : 0, UT : 6,		CONFIG : 'N U T, 0, 0, 0',
	X =  -3.435  mm,	Y =   -592.515  mm,	Z =   -235.802  mm,
	W =  90.000 deg,	P =   0.000 deg,	R =   90.000 deg
};
P[1126]{
   GP1:
	UF : 0, UT : 6,		CONFIG : 'N U T, 0, 0, 0',
	X =  -2.904  mm,	Y =   -593.281  mm,	Z =   -236.015  mm,
	W =  90.000 deg,	P =   0.000 deg,	R =   90.000 deg
};
P[1127]{
   GP1:
	UF : 0, UT : 6,		CONFIG : 'N U T, 0, 0, 0',
	X =  -2.619  mm,	Y =   -593.942  mm,	Z =   -235.783  mm,
	W =  90.000 deg,	P =   0.000 deg,	R =   90.000 deg
};
P[1128]{
   GP1:
	UF : 0, UT : 6,		CONFIG : 'N U T, 0, 0, 0',
	X =  -1.898  mm,	Y =   -594.885  mm,	Z =   -236.212  mm,
	W =  90.000 deg,	P =   0.000 deg,	R =   90.000 deg
};
P[1129]{
   GP1:
	UF : 0, UT : 6,		CONFIG : 'N U T, 0, 0, 0',
	X =  -1.390  mm,	Y =   -595.855  mm,	Z =   -236.087  mm,
	W =  90.000 deg,	P =   0.000 deg,	R =   90.000 deg
};
P[1130]{
   GP1:
	UF : 0, UT : 6,		CONFIG : 'N U T, 0, 0, 0',
	X =  -0.921  mm,	Y =   -596.565  mm,	Z =   -236.226  mm,
	W =  90.000 deg,	P =   0.000 deg,	R =   90.000 deg
};
P[1131]{
   GP1:
	UF : 0, UT : 6,		CONFIG : 'N U T, 0, 0, 0',
	X =  1.002  mm,	Y =   -599.892  mm,	Z =   -236.234  mm,
	W =  90.000 deg,	P =   0.000 deg,	R =   90.000 deg
};
P[1132]{
   GP1:
	UF : 0, UT : 6,		CONFIG : 'N U T, 0, 0, 0',
	X =  1.718  mm,	Y =   -601.286  mm,	Z =   -236.017  mm,
	W =  90.000 deg,	P =   0.000 deg,	R =   90.000 deg
};
P[1133]{
   GP1:
	UF : 0, UT : 6,		CONFIG : 'N U T, 0, 0, 0',
	X =  2.977  mm,	Y =   -603.431  mm,	Z =   -236.064  mm,
	W =  90.000 deg,	P =   0.000 deg,	R =   90.000 deg
};
P[1134]{
   GP1:
	UF : 0, UT : 6,		CONFIG : 'N U T, 0, 0, 0',
	X =  4.541  mm,	Y =   -606.107  mm,	Z =   -236.111  mm,
	W =  90.000 deg,	P =   0.000 deg,	R =   90.000 deg
};
P[1135]{
   GP1:
	UF : 0, UT : 6,		CONFIG : 'N U T, 0, 0, 0',
	X =  5.050  mm,	Y =   -607.189  mm,	Z =   -235.833  mm,
	W =  90.000 deg,	P =   0.000 deg,	R =   90.000 deg
};
P[1136]{
   GP1:
	UF : 0, UT : 6,		CONFIG : 'N U T, 0, 0, 0',
	X =  5.476  mm,	Y =   -607.794  mm,	Z =   -236.015  mm,
	W =  90.000 deg,	P =   0.000 deg,	R =   90.000 deg
};
P[1137]{
   GP1:
	UF : 0, UT : 6,		CONFIG : 'N U T, 0, 0, 0',
	X =  5.783  mm,	Y =   -608.399  mm,	Z =   -235.916  mm,
	W =  90.000 deg,	P =   0.000 deg,	R =   90.000 deg
};
P[1138]{
   GP1:
	UF : 0, UT : 6,		CONFIG : 'N U T, 0, 0, 0',
	X =  6.851  mm,	Y =   -610.071  mm,	Z =   -236.162  mm,
	W =  90.000 deg,	P =   0.000 deg,	R =   90.000 deg
};
P[1139]{
   GP1:
	UF : 0, UT : 6,		CONFIG : 'N U T, 0, 0, 0',
	X =  8.250  mm,	Y =   -612.740  mm,	Z =   -235.818  mm,
	W =  90.000 deg,	P =   0.000 deg,	R =   90.000 deg
};
P[1140]{
   GP1:
	UF : 0, UT : 6,		CONFIG : 'N U T, 0, 0, 0',
	X =  8.878  mm,	Y =   -613.702  mm,	Z =   -235.993  mm,
	W =  90.000 deg,	P =   0.000 deg,	R =   90.000 deg
};
P[1141]{
   GP1:
	UF : 0, UT : 6,		CONFIG : 'N U T, 0, 0, 0',
	X =  9.654  mm,	Y =   -614.927  mm,	Z =   -236.163  mm,
	W =  90.000 deg,	P =   0.000 deg,	R =   90.000 deg
};
P[1142]{
   GP1:
	UF : 0, UT : 6,		CONFIG : 'N U T, 0, 0, 0',
	X =  10.472  mm,	Y =   -616.364  mm,	Z =   -236.133  mm,
	W =  90.000 deg,	P =   0.000 deg,	R =   90.000 deg
};
P[1143]{
   GP1:
	UF : 0, UT : 6,		CONFIG : 'N U T, 0, 0, 0',
	X =  12.417  mm,	Y =   -619.743  mm,	Z =   -236.117  mm,
	W =  90.000 deg,	P =   0.000 deg,	R =   90.000 deg
};
P[1144]{
   GP1:
	UF : 0, UT : 6,		CONFIG : 'N U T, 0, 0, 0',
	X =  13.577  mm,	Y =   -621.654  mm,	Z =   -236.254  mm,
	W =  90.000 deg,	P =   0.000 deg,	R =   90.000 deg
};
P[1145]{
   GP1:
	UF : 0, UT : 6,		CONFIG : 'N U T, 0, 0, 0',
	X =  14.036  mm,	Y =   -622.574  mm,	Z =   -236.080  mm,
	W =  90.000 deg,	P =   0.000 deg,	R =   90.000 deg
};
P[1146]{
   GP1:
	UF : 0, UT : 6,		CONFIG : 'N U T, 0, 0, 0',
	X =  14.516  mm,	Y =   -623.470  mm,	Z =   -235.990  mm,
	W =  90.000 deg,	P =   0.000 deg,	R =   90.000 deg
};
P[1147]{
   GP1:
	UF : 0, UT : 6,		CONFIG : 'N U T, 0, 0, 0',
	X =  14.935  mm,	Y =   -624.158  mm,	Z =   -236.043  mm,
	W =  90.000 deg,	P =   0.000 deg,	R =   90.000 deg
};
P[1148]{
   GP1:
	UF : 0, UT : 6,		CONFIG : 'N U T, 0, 0, 0',
	X =  18.331  mm,	Y =   -630.229  mm,	Z =   -235.777  mm,
	W =  90.000 deg,	P =   0.000 deg,	R =   90.000 deg
};
P[1149]{
   GP1:
